C05443=1098.967,27.452,444.995,176.228,15.026,151.970
C05444=1098.962,27.202,445.009,176.226,15.025,151.971
C05445=1098.956,26.952,445.024,176.224,15.025,151.971
C05446=1098.951,26.703,445.039,176.221,15.024,151.971
C05447=1098.944,26.454,445.054,176.219,15.023,151.972
C05448=1098.939,26.204,445.069,176.217,15.022,151.972
C05449=1098.933,25.955,445.084,176.215,15.022,151.972
C05450=1098.927,25.705,445.098,176.212,15.021,151.973
C05451=1098.922,25.455,445.113,176.210,15.020,151.973
C05452=1098.916,25.206,445.128,176.208,15.020,151.973
C05453=1098.910,24.957,445.143,176.206,15.019,151.974
C05454=1098.904,24.708,445.157,176.203,15.018,151.974
C05455=1098.899,24.458,445.172,176.201,15.018,151.974
C05456=1098.893,24.208,445.187,176.199,15.017,151.975
C05457=1098.887,23.959,445.201,176.197,15.016,151.975
C05458=1098.881,23.709,445.217,176.194,15.015,151.975
C05459=1098.876,23.460,445.231,176.192,15.015,151.976
C05460=1098.869,23.210,445.246,176.190,15.014,151.976
C05461=1098.863,22.961,445.260,176.188,15.013,151.976
C05462=1098.858,22.712,445.276,176.186,15.012,151.976
C05463=1098.852,22.461,445.290,176.183,15.012,151.977
C05464=1098.847,22.213,445.304,176.182,15.011,151.977
C05465=1098.841,21.963,445.320,176.180,15.010,151.977
C05466=1098.835,21.713,445.334,176.177,15.009,151.978
C05467=1098.830,21.464,445.348,176.175,15.009,151.978
C05468=1098.823,21.214,445.363,176.173,15.008,151.979
C05469=1098.819,20.964,445.378,176.171,15.008,151.979
C05470=1098.813,20.716,445.392,176.168,15.006,151.979
C05471=1098.806,20.466,445.407,176.166,15.006,151.979
C05472=1098.801,20.216,445.421,176.164,15.005,151.980
C05473=1098.795,19.967,445.436,176.162,15.005,151.980
C05474=1098.789,19.717,445.451,176.159,15.004,151.980
C05475=1098.784,19.468,445.465,176.157,15.003,151.981
C05476=1098.778,19.218,445.480,176.155,15.002,151.981
C05477=1098.772,18.969,445.495,176.153,15.002,151.981
C05478=1098.766,18.719,445.509,176.151,15.001,151.982
C05479=1098.760,18.470,445.523,176.149,15.000,151.982
C05480=1098.755,18.220,445.538,176.147,14.999,151.982
C05481=1098.749,17.970,445.553,176.145,14.999,151.983
C05482=1098.743,17.721,445.567,176.143,14.998,151.983
C05483=1098.738,17.472,445.581,176.140,14.997,151.983
C05484=1098.731,17.222,445.596,176.138,14.996,151.984
C05485=1098.726,16.973,445.610,176.136,14.996,151.984
C05486=1098.720,16.724,445.625,176.134,14.995,151.984
C05487=1098.714,16.473,445.639,176.131,14.994,151.985
C05488=1098.709,16.224,445.654,176.129,14.993,151.985
C05489=1098.702,15.952,445.669,176.127,14.993,151.985
C05490=1098.696,15.680,445.685,176.125,14.992,151.985
C05491=1098.690,15.408,445.700,176.123,14.991,151.986
C05492=1098.684,15.136,445.716,176.120,14.991,151.986
C05493=1098.678,14.886,445.731,176.118,14.989,151.986
C05494=1098.672,14.637,445.745,176.116,14.988,151.987
C05495=1098.666,14.388,445.759,176.114,14.988,151.987
C05496=1098.660,14.137,445.773,176.112,14.987,151.987
C05497=1098.655,13.889,445.788,176.109,14.986,151.988
C05498=1098.649,13.639,445.802,176.107,14.985,151.988
C05499=1098.643,13.389,445.817,176.105,14.985,151.988
C05500=1098.637,13.140,445.831,176.103,14.984,151.989
C05501=1098.631,12.891,445.845,176.101,14.984,151.989
C05502=1098.625,12.640,445.860,176.098,14.983,151.989
C05503=1098.620,12.391,445.873,176.097,14.982,151.990
C05504=1098.614,12.142,445.888,176.095,14.981,151.990
C05505=1098.608,11.892,445.902,176.092,14.981,151.990
C05506=1098.602,11.642,445.915,176.091,14.980,151.990
C05507=1098.596,11.393,445.930,176.088,14.979,151.991
C05508=1098.590,11.143,445.944,176.086,14.978,151.991
C05509=1098.584,10.894,445.959,176.084,14.978,151.991
C05510=1098.579,10.645,445.973,176.082,14.977,151.992
C05511=1098.573,10.394,445.987,176.080,14.976,151.992
C05512=1098.567,10.145,446.002,176.077,14.975,151.992
C05513=1098.561,9.896,446.015,176.075,14.975,151.993
C05514=1098.556,9.646,446.029,176.073,14.974,151.993
C05515=1098.550,9.397,446.044,176.072,14.973,151.993
C05516=1098.543,9.147,446.057,176.070,14.972,151.993
C05517=1098.538,8.898,446.071,176.067,14.972,151.994
C05518=1098.532,8.648,446.085,176.065,14.971,151.994
C05519=1098.526,8.399,446.100,176.063,14.970,151.994
C05520=1098.520,8.149,446.114,176.061,14.969,151.995
C05521=1098.515,7.899,446.128,176.059,14.969,151.995
C05522=1098.510,7.650,446.142,176.056,14.968,151.995
C05523=1098.502,7.400,446.156,176.054,14.967,151.996
C05524=1098.497,7.151,446.170,176.052,14.966,151.996
C05525=1098.491,6.901,446.184,176.051,14.965,151.996
C05526=1098.486,6.652,446.198,176.048,14.965,151.997
C05527=1098.480,6.402,446.213,176.046,14.964,151.997
C05528=1098.474,6.153,446.227,176.044,14.963,151.997
C05529=1098.469,5.903,446.240,176.042,14.962,151.997
C05530=1098.462,5.654,446.254,176.040,14.962,151.998
C05531=1098.457,5.404,446.268,176.038,14.961,151.998
C05532=1098.451,5.154,446.282,176.036,14.961,151.998
C05533=1098.445,4.905,446.296,176.033,14.959,151.999
C05534=1098.440,4.655,446.310,176.031,14.958,151.999
C05535=1098.433,4.406,446.323,176.030,14.958,151.999
C05536=1098.428,4.156,446.337,176.028,14.957,151.999
C05537=1098.422,3.907,446.351,176.026,14.956,152.000
C05538=1098.416,3.657,446.365,176.023,14.955,152.000
C05539=1098.411,3.408,446.380,176.021,14.955,152.000
C05540=1098.404,3.158,446.393,176.019,14.954,152.001
C05541=1098.399,2.909,446.407,176.017,14.953,152.001
C05542=1098.393,2.659,446.421,176.015,14.952,152.001
C05543=1098.388,2.410,446.435,176.014,14.952,152.001
C05544=1098.382,2.160,446.449,176.011,14.950,152.002
C05545=1098.376,1.910,446.462,176.009,14.950,152.002
C05546=1098.370,1.661,446.476,176.007,14.949,152.002
C05547=1098.365,1.411,446.490,176.005,14.949,152.003
C05548=1098.359,1.161,446.504,176.003,14.948,152.003
C05549=1098.353,0.912,446.517,176.001,14.947,152.003
C05550=1098.348,0.663,446.531,175.998,14.946,152.003
C05551=1098.342,0.413,446.545,175.997,14.945,152.004
C05552=1098.337,0.163,446.559,175.995,14.944,152.004
C05553=1098.330,-0.107,446.574,175.993,14.943,152.004
C05554=1098.324,-0.377,446.588,175.990,14.942,152.004
C05555=1098.317,-0.646,446.604,175.988,14.941,152.005
C05556=1098.311,-0.917,446.619,175.986,14.941,152.005
C05557=1098.305,-1.166,446.632,175.983,14.940,152.005
C05558=1098.300,-1.416,446.646,175.982,14.939,152.006
C05559=1098.294,-1.665,446.660,175.980,14.938,152.006
C05560=1098.289,-1.915,446.673,175.978,14.938,152.006
C05561=1098.283,-2.165,446.686,175.976,14.937,152.006
C05562=1098.277,-2.414,446.700,175.974,14.936,152.007
C05563=1098.272,-2.664,446.714,175.971,14.935,152.007
C05564=1098.265,-2.913,446.727,175.970,14.934,152.007
C05565=1098.260,-3.163,446.741,175.968,14.933,152.007
C05566=1098.255,-3.412,446.755,175.966,14.932,152.008
C05567=1098.248,-3.661,446.768,175.964,14.932,152.008
C05568=1098.242,-3.912,446.782,175.962,14.931,152.008
C05569=1098.236,-4.161,446.796,175.960,14.930,152.008
C05570=1098.231,-4.411,446.810,175.957,14.929,152.009
C05571=1098.225,-4.660,446.822,175.955,14.929,152.009
C05572=1098.219,-4.910,446.836,175.953,14.928,152.009
C05573=1098.213,-5.159,446.849,175.952,14.927,152.010
C05574=1098.207,-5.409,446.863,175.950,14.926,152.010
C05575=1098.201,-5.658,446.876,175.948,14.926,152.010
C05576=1098.196,-5.908,446.890,175.946,14.925,152.010
C05577=1098.190,-6.157,446.904,175.943,14.924,152.011
C05578=1098.184,-6.408,446.917,175.941,14.923,152.011
C05579=1098.178,-6.657,446.930,175.940,14.922,152.011
C05580=1098.172,-6.907,446.944,175.938,14.921,152.012
C05581=1098.166,-7.156,446.958,175.935,14.921,152.012
C05582=1098.160,-7.406,446.971,175.934,14.920,152.012
C05583=1098.155,-7.655,446.984,175.932,14.920,152.013
C05584=1098.149,-7.905,446.998,175.930,14.919,152.013
C05585=1098.143,-8.154,447.011,175.927,14.917,152.013
C05586=1098.137,-8.404,447.025,175.925,14.917,152.013
C05587=1098.131,-8.653,447.038,175.923,14.916,152.014
C05588=1098.126,-8.903,447.051,175.922,14.915,152.014
C05589=1098.120,-9.153,447.065,175.920,14.915,152.014
C05590=1098.114,-9.402,447.078,175.918,14.914,152.014
C05591=1098.108,-9.652,447.091,175.916,14.913,152.015
C05592=1098.102,-9.901,447.104,175.914,14.912,152.015
C05593=1098.097,-10.151,447.118,175.911,14.911,152.015
C05594=1098.090,-10.400,447.131,175.909,14.910,152.015
C05595=1098.085,-10.650,447.145,175.908,14.909,152.016
C05596=1098.079,-10.900,447.158,175.906,14.909,152.016
C05597=1098.074,-11.149,447.172,175.904,14.908,152.016
C05598=1098.068,-11.399,447.184,175.902,14.907,152.016
C05599=1098.061,-11.648,447.198,175.900,14.906,152.017
C05600=1098.056,-11.898,447.211,175.898,14.906,152.017
C05601=1098.050,-12.148,447.224,175.896,14.904,152.017
C05602=1098.045,-12.397,447.238,175.894,14.904,152.018
C05603=1098.038,-12.647,447.251,175.892,14.903,152.018
C05604=1098.033,-12.896,447.264,175.890,14.902,152.018
C05605=1098.027,-13.146,447.278,175.888,14.901,152.018
C05606=1098.021,-13.396,447.290,175.886,14.901,152.019
C05607=1098.016,-13.645,447.304,175.884,14.900,152.019
C05608=1098.009,-13.895,447.317,175.882,14.899,152.019
C05609=1098.004,-14.144,447.329,175.881,14.898,152.019
C05610=1097.999,-14.393,447.343,175.878,14.897,152.020
C05611=1097.993,-14.643,447.356,175.876,14.896,152.020
C05612=1097.987,-14.893,447.369,175.874,14.896,152.020
C05613=1097.981,-15.143,447.382,175.872,14.895,152.020
C05614=1097.975,-15.392,447.395,175.870,14.894,152.021
C05615=1097.969,-15.641,447.409,175.868,14.893,152.021
C05616=1097.963,-15.891,447.421,175.867,14.893,152.021
C05617=1097.957,-16.160,447.436,175.865,14.892,152.021
C05618=1097.950,-16.428,447.449,175.862,14.891,152.022
C05619=1097.944,-16.697,447.464,175.860,14.890,152.022
C05620=1097.938,-16.965,447.477,175.858,14.890,152.022
C05621=1097.932,-17.214,447.491,175.856,14.889,152.023
C05622=1097.927,-17.465,447.504,175.854,14.888,152.023
C05623=1097.920,-17.714,447.517,175.852,14.887,152.023
C05624=1097.914,-17.964,447.530,175.850,14.886,152.023
C05625=1097.908,-18.213,447.543,175.848,14.885,152.024
C05626=1097.902,-18.463,447.556,175.846,14.885,152.024
C05627=1097.897,-18.712,447.569,175.844,14.884,152.024
C05628=1097.892,-18.962,447.582,175.842,14.883,152.025
C05629=1097.885,-19.211,447.595,175.840,14.882,152.025
C05630=1097.879,-19.461,447.607,175.838,14.882,152.025
C05631=1097.873,-19.710,447.621,175.837,14.881,152.025
C05632=1097.867,-19.960,447.633,175.835,14.880,152.026
C05633=1097.862,-20.210,447.646,175.833,14.879,152.026
C05634=1097.856,-20.459,447.660,175.831,14.879,152.026
C05635=1097.850,-20.709,447.672,175.829,14.878,152.026
C05636=1097.844,-20.959,447.685,175.827,14.877,152.026
C05637=1097.839,-21.208,447.698,175.825,14.875,152.027
C05638=1097.833,-21.458,447.710,175.823,14.875,152.027
C05639=1097.827,-21.707,447.724,175.821,14.874,152.027
C05640=1097.821,-21.957,447.737,175.819,14.873,152.027
C05641=1097.815,-22.206,447.750,175.817,14.872,152.028
C05642=1097.809,-22.456,447.762,175.815,14.872,152.028
C05643=1097.803,-22.706,447.775,175.814,14.871,152.028
C05644=1097.798,-22.955,447.788,175.812,14.870,152.029
C05645=1097.792,-23.205,447.800,175.810,14.869,152.029
C05646=1097.786,-23.455,447.813,175.808,14.869,152.029
C05647=1097.780,-23.704,447.827,175.806,14.868,152.029
C05648=1097.774,-23.954,447.839,175.804,14.867,152.030
C05649=1097.768,-24.204,447.852,175.802,14.866,152.030
C05650=1097.763,-24.453,447.864,175.800,14.866,152.030
C05651=1097.757,-24.702,447.877,175.798,14.864,152.030
C05652=1097.751,-24.952,447.890,175.796,14.864,152.031
C05653=1097.745,-25.202,447.903,175.794,14.863,152.031
C05654=1097.739,-25.451,447.916,175.792,14.862,152.031
C05655=1097.734,-25.701,447.928,175.790,14.861,152.031
C05656=1097.728,-25.951,447.941,175.789,14.860,152.032
C05657=1097.723,-26.201,447.954,175.787,14.859,152.032
C05658=1097.717,-26.450,447.966,175.785,14.859,152.032
C05659=1097.710,-26.700,447.980,175.783,14.858,152.032
C05660=1097.705,-26.949,447.992,175.781,14.857,152.033
C05661=1097.699,-27.199,448.004,175.779,14.857,152.033
C05662=1097.693,-27.449,448.017,175.777,14.856,152.033
C05663=1097.687,-27.698,448.030,175.776,14.855,152.033
C05664=1097.681,-27.948,448.043,175.774,14.854,152.034
C05665=1097.676,-28.197,448.055,175.772,14.854,152.034
C05666=1097.669,-28.447,448.067,175.770,14.853,152.034
C05667=1097.663,-28.696,448.079,175.768,14.852,152.034
C05668=1097.657,-28.946,448.093,175.766,14.851,152.035
C05669=1097.651,-29.196,448.105,175.764,14.851,152.035
C05670=1097.646,-29.445,448.117,175.762,14.850,152.035
C05671=1097.640,-29.695,448.130,175.760,14.849,152.035
C05672=1097.634,-29.945,448.142,175.759,14.848,152.036
C05673=1097.628,-30.194,448.155,175.757,14.848,152.036
C05674=1097.622,-30.444,448.168,175.754,14.846,152.036
C05675=1097.617,-30.693,448.181,175.752,14.846,152.036
C05676=1097.611,-30.943,448.193,175.750,14.845,152.037
C05677=1097.604,-31.192,448.205,175.748,14.844,152.037
C05678=1097.598,-31.442,448.218,175.747,14.843,152.037
C05679=1097.593,-31.691,448.230,175.745,14.842,152.037
C05680=1097.587,-31.941,448.242,175.743,14.841,152.038
C05681=1097.581,-32.209,448.256,175.741,14.841,152.038
C05682=1097.575,-32.477,448.269,175.739,14.840,152.038
C05683=1097.567,-32.744,448.283,175.737,14.839,152.038
C05684=1097.561,-33.012,448.296,175.736,14.839,152.039
C05685=1097.556,-33.261,448.308,175.734,14.838,152.039
C05686=1097.550,-33.511,448.320,175.732,14.837,152.039
C05687=1097.544,-33.761,448.333,175.730,14.836,152.039
C05688=1097.538,-34.010,448.346,175.728,14.836,152.040
C05689=1097.532,-34.259,448.358,175.726,14.835,152.040
C05690=1097.526,-34.509,448.370,175.724,14.834,152.040
C05691=1097.520,-34.759,448.383,175.722,14.833,152.040
C05692=1097.515,-35.008,448.395,175.721,14.833,152.041
C05693=1097.509,-35.258,448.408,175.719,14.832,152.041
C05694=1097.503,-35.508,448.420,175.717,14.831,152.041
C05695=1097.497,-35.758,448.431,175.715,14.830,152.042
C05696=1097.492,-36.007,448.444,175.713,14.830,152.042
C05697=1097.486,-36.257,448.456,175.711,14.829,152.042
C05698=1097.480,-36.507,448.469,175.709,14.827,152.042
C05699=1097.474,-36.756,448.481,175.707,14.826,152.042
C05700=1097.468,-37.006,448.493,175.705,14.826,152.043
C05701=1097.462,-37.256,448.505,175.703,14.825,152.043
C05702=1097.457,-37.505,448.518,175.701,14.824,152.043
C05703=1097.451,-37.755,448.530,175.699,14.823,152.044
C05704=1097.445,-38.005,448.543,175.698,14.823,152.044
C05705=1097.439,-38.254,448.555,175.696,14.822,152.044
C05706=1097.433,-38.503,448.567,175.695,14.822,152.044
C05707=1097.427,-38.753,448.579,175.693,14.821,152.044
C05708=1097.422,-39.003,448.592,175.691,14.820,152.045
C05709=1097.415,-39.253,448.603,175.689,14.819,152.045
C05710=1097.409,-39.503,448.615,175.687,14.818,152.045
C05711=1097.404,-39.752,448.628,175.685,14.818,152.045
C05712=1097.397,-40.001,448.640,175.684,14.817,152.046
C05713=1097.391,-40.251,448.652,175.682,14.816,152.046
C05714=1097.386,-40.500,448.664,175.680,14.816,152.046
C05715=1097.379,-40.750,448.676,175.678,14.815,152.046
C05716=1097.374,-41.000,448.688,175.676,14.814,152.047
C05717=1097.369,-41.250,448.700,175.674,14.813,152.047
C05718=1097.362,-41.499,448.712,175.672,14.813,152.047
C05719=1097.356,-41.749,448.725,175.670,14.812,152.047
C05720=1097.350,-41.998,448.736,175.669,14.811,152.048
C05721=1097.344,-42.248,448.749,175.667,14.810,152.048
C05722=1097.338,-42.498,448.761,175.665,14.810,152.048
C05723=1097.332,-42.747,448.772,175.663,14.809,152.049
C05724=1097.326,-42.997,448.785,175.661,14.808,152.049
C05725=1097.321,-43.247,448.797,175.659,14.807,152.049
C05726=1097.315,-43.497,448.808,175.657,14.807,152.049
C05727=1097.309,-43.746,448.821,175.656,14.806,152.049
C05728=1097.303,-43.995,448.832,175.654,14.805,152.050
C05729=1097.297,-44.245,448.845,175.652,14.804,152.050
C05730=1097.291,-44.496,448.857,175.650,14.803,152.050
C05731=1097.285,-44.745,448.868,175.648,14.803,152.050
C05732=1097.279,-44.994,448.881,175.646,14.802,152.051
C05733=1097.273,-45.243,448.893,175.644,14.801,152.051
C05734=1097.268,-45.494,448.904,175.643,14.800,152.051
C05735=1097.261,-45.743,448.916,175.641,14.800,152.052
C05736=1097.256,-45.993,448.929,175.639,14.799,152.052
C05737=1097.250,-46.243,448.940,175.637,14.798,152.052
C05738=1097.244,-46.492,448.952,175.635,14.797,152.052
C05739=1097.238,-46.742,448.965,175.634,14.797,152.053
C05740=1097.232,-46.992,448.976,175.632,14.797,152.053
C05741=1097.227,-47.241,448.988,175.630,14.795,152.053
C05742=1097.220,-47.491,449.000,175.629,14.795,152.053
C05743=1097.215,-47.741,449.011,175.627,14.794,152.053
C05744=1097.208,-47.990,449.023,175.625,14.793,152.054
C05745=1097.202,-48.258,449.036,175.623,14.792,152.054
C05746=1097.196,-48.526,449.049,175.621,14.792,152.054
C05747=1097.190,-48.794,449.062,175.619,14.791,152.054
C05748=1097.183,-49.061,449.074,175.616,14.790,152.055
C05749=1097.178,-49.312,449.086,175.615,14.790,152.055
C05750=1097.172,-49.561,449.098,175.614,14.789,152.055
C05751=1097.166,-49.810,449.110,175.612,14.788,152.055
C05752=1097.160,-50.060,449.121,175.610,14.787,152.056
C05753=1097.154,-50.310,449.134,175.608,14.787,152.056
C05754=1097.148,-50.559,449.145,175.606,14.786,152.056
C05755=1097.142,-50.809,449.157,175.604,14.785,152.057
C05756=1097.136,-51.059,449.168,175.602,14.784,152.057
C05757=1097.130,-51.308,449.180,175.600,14.784,152.057
C05758=1097.124,-51.558,449.193,175.598,14.783,152.057
C05759=1097.118,-51.808,449.203,175.597,14.782,152.058
C05760=1097.112,-52.057,449.215,175.595,14.782,152.058
C05761=1097.106,-52.308,449.227,175.593,14.781,152.058
C05762=1097.100,-52.557,449.239,175.592,14.781,152.058
C05763=1097.094,-52.807,449.250,175.590,14.780,152.059
C05764=1097.089,-53.056,449.262,175.588,14.779,152.059
C05765=1097.082,-53.306,449.273,175.586,14.778,152.059
C05766=1097.076,-53.555,449.285,175.584,14.778,152.059
C05767=1097.070,-53.805,449.296,175.582,14.777,152.060
C05768=1097.064,-54.055,449.309,175.580,14.776,152.060
C05769=1097.058,-54.305,449.320,175.579,14.776,152.060
C05770=1097.051,-54.554,449.332,175.577,14.775,152.060
C05771=1097.046,-54.804,449.343,175.575,14.774,152.061
C05772=1097.040,-55.054,449.355,175.573,14.773,152.061
C05773=1097.034,-55.303,449.366,175.572,14.773,152.061
C05774=1097.027,-55.553,449.378,175.570,14.773,152.061
C05775=1097.022,-55.802,449.389,175.568,14.772,152.062
C05776=1097.016,-56.052,449.401,175.566,14.771,152.062
C05777=1097.010,-56.301,449.412,175.564,14.770,152.062
C05778=1097.004,-56.552,449.424,175.562,14.770,152.063
C05779=1096.998,-56.801,449.435,175.561,14.769,152.063
C05780=1096.992,-57.051,449.447,175.559,14.768,152.063
C05781=1096.986,-57.300,449.459,175.557,14.767,152.063
C05782=1096.980,-57.550,449.470,175.556,14.767,152.064
C05783=1096.974,-57.799,449.481,175.554,14.767,152.064
C05784=1096.968,-58.049,449.493,175.552,14.766,152.064
C05785=1096.962,-58.299,449.504,175.550,14.765,152.064
C05786=1096.956,-58.549,449.516,175.548,14.764,152.064
C05787=1096.950,-58.798,449.527,175.547,14.763,152.065
C05788=1096.944,-59.048,449.538,175.545,14.762,152.065
C05789=1096.938,-59.297,449.550,175.543,14.762,152.065
C05790=1096.932,-59.548,449.562,175.542,14.762,152.065
C05791=1096.926,-59.797,449.573,175.540,14.761,152.066
C05792=1096.920,-60.047,449.584,175.538,14.760,152.066
C05793=1096.914,-60.296,449.595,175.536,14.759,152.066
C05794=1096.908,-60.547,449.607,175.534,14.759,152.066
C05795=1096.902,-60.796,449.619,175.532,14.758,152.067
C05796=1096.896,-61.046,449.630,175.530,14.757,152.067
C05797=1096.890,-61.295,449.641,175.529,14.757,152.067
C05798=1096.884,-61.544,449.652,175.527,14.756,152.068
C05799=1096.878,-61.794,449.664,175.526,14.756,152.068
C05800=1096.873,-62.044,449.675,175.524,14.755,152.068
C05801=1096.866,-62.294,449.686,175.522,14.754,152.068
C05802=1096.860,-62.543,449.698,175.520,14.753,152.069
C05803=1096.855,-62.793,449.709,175.518,14.753,152.069
C05804=1096.848,-63.043,449.720,175.516,14.752,152.069
C05805=1096.842,-63.292,449.731,175.515,14.752,152.069
C05806=1096.837,-63.542,449.744,175.513,14.751,152.070
C05807=1096.831,-63.792,449.754,175.511,14.750,152.070
C05808=1096.825,-64.042,449.766,175.509,14.750,152.070
C05809=1096.818,-64.310,449.777,175.507,14.749,152.070
C05810=1096.812,-64.579,449.790,175.506,14.748,152.071
C05811=1096.805,-64.849,449.801,175.504,14.748,152.071
C05812=1096.799,-65.118,449.814,175.502,14.747,152.071
C05813=1096.793,-65.368,449.825,175.500,14.746,152.071
C05814=1096.787,-65.618,449.836,175.498,14.745,152.072
C05815=1096.781,-65.867,449.848,175.496,14.745,152.072
C05816=1096.775,-66.117,449.859,175.495,14.745,152.072
C05817=1096.770,-66.367,449.871,175.493,14.744,152.072
C05818=1096.764,-66.616,449.881,175.491,14.743,152.073
C05819=1096.758,-66.866,449.893,175.489,14.742,152.073
C05820=1096.752,-67.116,449.904,175.488,14.742,152.073
C05821=1096.746,-67.365,449.914,175.486,14.741,152.074
C05822=1096.740,-67.615,449.926,175.485,14.741,152.074
C05823=1096.734,-67.865,449.937,175.483,14.740,152.074
C05824=1096.728,-68.114,449.948,175.481,14.739,152.074
C05825=1096.722,-68.364,449.959,175.479,14.739,152.075
C05826=1096.716,-68.614,449.970,175.477,14.738,152.075
C05827=1096.710,-68.863,449.981,175.475,14.737,152.075
C05828=1096.705,-69.114,449.993,175.474,14.737,152.075
C05829=1096.699,-69.363,450.004,175.472,14.736,152.076
C05830=1096.693,-69.613,450.015,175.470,14.736,152.076
C05831=1096.687,-69.863,450.026,175.468,14.735,152.076
C05832=1096.681,-70.112,450.038,175.467,14.734,152.076
C05833=1096.675,-70.361,450.048,175.465,14.733,152.077
C05834=1096.669,-70.611,450.059,175.464,14.733,152.077
C05835=1096.663,-70.861,450.071,175.462,14.733,152.077
C05836=1096.657,-71.110,450.081,175.460,14.732,152.077
C05837=1096.652,-71.360,450.092,175.458,14.731,152.078
C05838=1096.645,-71.610,450.104,175.456,14.730,152.078
C05839=1096.639,-71.860,450.114,175.455,14.730,152.078
C05840=1096.634,-72.109,450.125,175.453,14.730,152.078
C05841=1096.628,-72.359,450.136,175.451,14.729,152.079
C05842=1096.622,-72.609,450.147,175.450,14.728,152.079
C05843=1096.616,-72.858,450.158,175.448,14.727,152.079
C05844=1096.610,-73.108,450.169,175.446,14.726,152.079
C05845=1096.604,-73.357,450.180,175.445,14.726,152.079
C05846=1096.599,-73.608,450.192,175.443,14.725,152.080
C05847=1096.593,-73.857,450.203,175.441,14.725,152.080
C05848=1096.587,-74.107,450.214,175.439,14.724,152.080
C05849=1096.581,-74.356,450.224,175.437,14.723,152.081
C05850=1096.575,-74.606,450.235,175.436,14.723,152.081
C05851=1096.569,-74.856,450.246,175.434,14.722,152.081
C05852=1096.563,-75.106,450.256,175.432,14.722,152.081
C05853=1096.557,-75.356,450.267,175.430,14.721,152.082
C05854=1096.551,-75.605,450.278,175.429,14.721,152.082
C05855=1096.546,-75.855,450.289,175.427,14.720,152.082
C05856=1096.539,-76.105,450.300,175.425,14.720,152.082
C05857=1096.533,-76.354,450.311,175.423,14.719,152.083
C05858=1096.527,-76.604,450.322,175.421,14.718,152.083
C05859=1096.521,-76.853,450.333,175.420,14.718,152.083
C05860=1096.515,-77.103,450.344,175.418,14.717,152.084
C05861=1096.509,-77.353,450.355,175.417,14.717,152.084
C05862=1096.503,-77.602,450.366,175.415,14.716,152.084
C05863=1096.497,-77.851,450.376,175.414,14.716,152.084
C05864=1096.491,-78.102,450.386,175.412,14.715,152.085
C05865=1096.485,-78.352,450.397,175.410,14.714,152.085
C05866=1096.479,-78.601,450.408,175.408,14.714,152.085
C05867=1096.474,-78.851,450.419,175.406,14.713,152.085
C05868=1096.467,-79.101,450.430,175.405,14.713,152.086
C05869=1096.461,-79.350,450.440,175.403,14.712,152.086
C05870=1096.455,-79.600,450.451,175.401,14.712,152.086
C05871=1096.450,-79.850,450.462,175.399,14.711,152.087
C05872=1096.443,-80.100,450.473,175.398,14.711,152.087
C05873=1096.436,-80.371,450.484,175.396,14.710,152.087
C05874=1096.430,-80.642,450.495,175.394,14.710,152.087
C05875=1096.424,-80.914,450.507,175.392,14.709,152.088
C05876=1096.417,-81.185,450.518,175.390,14.709,152.088
C05877=1096.411,-81.434,450.529,175.388,14.708,152.088
C05878=1096.405,-81.685,450.541,175.387,14.708,152.088
C05879=1096.398,-81.934,450.551,175.385,14.707,152.089
C05880=1096.393,-82.184,450.561,175.383,14.706,152.089
C05881=1096.387,-82.433,450.572,175.381,14.706,152.089
C05882=1096.380,-82.683,450.582,175.380,14.706,152.089
C05883=1096.374,-82.933,450.593,175.378,14.705,152.090
C05884=1096.369,-83.183,450.604,175.376,14.705,152.090
C05885=1096.362,-83.432,450.614,175.374,14.704,152.090
C05886=1096.356,-83.682,450.625,175.373,14.704,152.091
C05887=1096.350,-83.932,450.636,175.371,14.703,152.091
C05888=1096.344,-84.182,450.645,175.369,14.702,152.091
C05889=1096.338,-84.431,450.656,175.368,14.702,152.091
C05890=1096.331,-84.681,450.667,175.366,14.702,152.092
C05891=1096.325,-84.930,450.678,175.364,14.701,152.092
C05892=1096.320,-85.181,450.688,175.362,14.701,152.092
C05893=1096.313,-85.430,450.698,175.361,14.700,152.093
C05894=1096.308,-85.679,450.709,175.359,14.700,152.093
C05895=1096.301,-85.930,450.719,175.357,14.699,152.093
C05896=1096.295,-86.179,450.730,175.356,14.698,152.093
C05897=1096.289,-86.429,450.741,175.354,14.699,152.094
C05898=1096.283,-86.679,450.750,175.352,14.698,152.094
C05899=1096.278,-86.928,450.761,175.350,14.697,152.094
C05900=1096.270,-87.178,450.772,175.348,14.696,152.095
C05901=1096.265,-87.428,450.782,175.347,14.696,152.095
C05902=1096.259,-87.677,450.793,175.346,14.696,152.095
C05903=1096.253,-87.927,450.803,175.344,14.695,152.095
C05904=1096.247,-88.177,450.813,175.342,14.695,152.096
C05905=1096.240,-88.427,450.824,175.340,14.695,152.096
C05906=1096.235,-88.676,450.835,175.338,14.694,152.096
C05907=1096.228,-88.926,450.845,175.337,14.694,152.097
C05908=1096.223,-89.175,450.855,175.335,14.693,152.097
C05909=1096.217,-89.426,450.866,175.334,14.692,152.097
C05910=1096.211,-89.675,450.876,175.332,14.692,152.097
C05911=1096.205,-89.924,450.887,175.330,14.692,152.098
C05912=1096.198,-90.175,450.897,175.328,14.691,152.098
C05913=1096.193,-90.424,450.908,175.326,14.691,152.098
C05914=1096.186,-90.674,450.917,175.325,14.690,152.098
C05915=1096.181,-90.923,450.928,175.323,14.690,152.099
C05916=1096.174,-91.173,450.938,175.322,14.689,152.099
C05917=1096.169,-91.423,450.948,175.320,14.689,152.099
C05918=1096.162,-91.672,450.959,175.318,14.689,152.100
C05919=1096.157,-91.922,450.969,175.316,14.688,152.100
C05920=1096.150,-92.172,450.980,175.315,14.687,152.100
C05921=1096.144,-92.422,450.990,175.313,14.687,152.100
C05922=1096.139,-92.672,451.001,175.312,14.686,152.101
C05923=1096.132,-92.921,451.010,175.309,14.686,152.101
C05924=1096.127,-93.171,451.021,175.308,14.686,152.101
C05925=1096.120,-93.421,451.031,175.306,14.685,152.102
C05926=1096.115,-93.670,451.041,175.304,14.685,152.102
C05927=1096.109,-93.920,451.051,175.303,14.684,152.102
C05928=1096.103,-94.169,451.062,175.301,14.684,152.102
C05929=1096.097,-94.419,451.072,175.299,14.684,152.103
C05930=1096.091,-94.669,451.082,175.298,14.683,152.103
C05931=1096.084,-94.919,451.092,175.296,14.683,152.103
C05932=1096.079,-95.169,451.102,175.294,14.682,152.104
C05933=1096.072,-95.418,451.113,175.293,14.682,152.104
C05934=1096.067,-95.669,451.123,175.291,14.681,152.104
C05935=1096.060,-95.918,451.133,175.289,14.681,152.104
C05936=1096.055,-96.168,451.143,175.288,14.681,152.105
C05937=1096.048,-96.441,451.155,175.286,14.680,152.105
C05938=1096.042,-96.714,451.166,175.284,14.679,152.105
C05939=1096.035,-96.988,451.176,175.282,14.679,152.106
C05940=1096.028,-97.262,451.187,175.280,14.678,152.106
C05941=1096.022,-97.512,451.198,175.279,14.678,152.106
C05942=1096.016,-97.762,451.208,175.277,14.678,152.106
C05943=1096.011,-98.012,451.218,175.275,14.677,152.107
C05944=1096.004,-98.261,451.228,175.274,14.677,152.107
C05945=1095.998,-98.511,451.238,175.272,14.677,152.107
C05946=1095.992,-98.761,451.249,175.270,14.676,152.108
C05947=1095.986,-99.011,451.259,175.269,14.676,152.108
C05948=1095.980,-99.260,451.268,175.267,14.675,152.108
C05949=1095.974,-99.510,451.279,175.266,14.675,152.109
C05950=1095.968,-99.760,451.289,175.263,14.675,152.109
C05951=1095.961,-100.009,451.298,175.262,14.674,152.109
C05952=1095.955,-100.259,451.308,175.260,14.674,152.109
C05953=1095.950,-100.509,451.319,175.259,14.674,152.110
C05954=1095.943,-100.759,451.328,175.256,14.673,152.110
C05955=1095.937,-101.008,451.339,175.255,14.673,152.110
C05956=1095.931,-101.258,451.349,175.253,14.673,152.111
C05957=1095.925,-101.508,451.358,175.252,14.672,152.111
C05958=1095.919,-101.757,451.369,175.250,14.672,152.111
C05959=1095.913,-102.007,451.379,175.248,14.671,152.112
C05960=1095.907,-102.257,451.388,175.247,14.671,152.112
C05961=1095.901,-102.506,451.399,175.245,14.671,152.112
C05962=1095.895,-102.756,451.408,175.243,14.670,152.112
C05963=1095.889,-103.006,451.418,175.242,14.670,152.113
C05964=1095.883,-103.255,451.429,175.240,14.670,152.113
C05965=1095.876,-103.505,451.438,175.239,14.670,152.113
C05966=1095.870,-103.755,451.448,175.237,14.669,152.114
C05967=1095.864,-104.005,451.458,175.235,14.669,152.114
C05968=1095.858,-104.255,451.468,175.233,14.669,152.114
C05969=1095.852,-104.504,451.478,175.232,14.668,152.115
C05970=1095.845,-104.754,451.488,175.230,14.668,152.115
C05971=1095.840,-105.004,451.498,175.229,14.667,152.115
C05972=1095.834,-105.253,451.508,175.226,14.667,152.115
C05973=1095.827,-105.503,451.518,175.225,14.667,152.116
C05974=1095.821,-105.753,451.527,175.223,14.666,152.116
C05975=1095.816,-106.003,451.537,175.221,14.666,152.116
C05976=1095.810,-106.253,451.547,175.220,14.666,152.117
C05977=1095.803,-106.502,451.557,175.218,14.665,152.117
C05978=1095.797,-106.752,451.567,175.217,14.666,152.117
C05979=1095.791,-107.002,451.576,175.215,14.665,152.118
C05980=1095.785,-107.251,451.586,175.213,14.664,152.118
C05981=1095.780,-107.501,451.596,175.211,14.665,152.118
C05982=1095.773,-107.750,451.606,175.210,14.664,152.118
C05983=1095.767,-108.000,451.616,175.208,14.664,152.119
C05984=1095.761,-108.250,451.625,175.206,14.664,152.119
C05985=1095.755,-108.500,451.635,175.205,14.663,152.119
C05986=1095.749,-108.749,451.644,175.203,14.663,152.120
C05987=1095.742,-108.999,451.654,175.201,14.663,152.120
C05988=1095.737,-109.249,451.665,175.200,14.662,152.120
C05989=1095.731,-109.498,451.674,175.198,14.662,152.121
C05990=1095.724,-109.748,451.684,175.197,14.662,152.121
C05991=1095.718,-109.998,451.693,175.195,14.661,152.121
C05992=1095.712,-110.248,451.703,175.193,14.661,152.122
C05993=1095.706,-110.498,451.713,175.191,14.661,152.122
C05994=1095.700,-110.747,451.722,175.190,14.660,152.122
C05995=1095.693,-110.997,451.732,175.188,14.661,152.123
C05996=1095.687,-111.247,451.741,175.186,14.660,152.123
C05997=1095.681,-111.496,451.752,175.185,14.660,152.123
C05998=1095.675,-111.746,451.761,175.183,14.660,152.123
C05999=1095.668,-111.996,451.771,175.181,14.659,152.124
C06000=1095.663,-112.246,451.781,175.180,14.659,152.124
C06001=1095.656,-112.509,451.791,175.178,14.659,152.124
C06002=1095.650,-112.774,451.801,175.176,14.659,152.125
C06003=1095.643,-113.037,451.811,175.174,14.658,152.125
C06004=1095.637,-113.301,451.821,175.173,14.658,152.125
C06005=1095.631,-113.550,451.831,175.171,14.658,152.126
C06006=1095.625,-113.800,451.840,175.169,14.657,152.126
C06007=1095.619,-114.050,451.850,175.168,14.658,152.126
C06008=1095.613,-114.300,451.859,175.166,14.657,152.127
C06009=1095.606,-114.550,451.869,175.165,14.657,152.127
C06010=1095.600,-114.799,451.879,175.163,14.657,152.127
C06011=1095.595,-115.049,451.888,175.161,14.656,152.128
C06012=1095.588,-115.298,451.897,175.159,14.656,152.128
C06013=1095.582,-115.548,451.907,175.157,14.656,152.128
C06014=1095.576,-115.798,451.917,175.156,14.656,152.129
C06015=1095.570,-116.048,451.926,175.154,14.655,152.129
C06016=1095.564,-116.298,451.936,175.153,14.655,152.129
C06017=1095.558,-116.547,451.945,175.151,14.655,152.130
C06018=1095.551,-116.797,451.955,175.150,14.655,152.130
C06019=1095.545,-117.047,451.964,175.147,14.655,152.130
C06020=1095.539,-117.297,451.974,175.146,14.654,152.130
C06021=1095.533,-117.546,451.983,175.144,14.654,152.131
C06022=1095.526,-117.796,451.992,175.143,14.654,152.131
C06023=1095.520,-118.045,452.002,175.141,14.654,152.132
C06024=1095.514,-118.295,452.011,175.139,14.653,152.132
C06025=1095.508,-118.545,452.021,175.137,14.654,152.132
C06026=1095.502,-118.794,452.030,175.136,14.653,152.132
C06027=1095.496,-119.044,452.040,175.134,14.653,152.133
C06028=1095.490,-119.294,452.049,175.132,14.653,152.133
C06029=1095.483,-119.544,452.059,175.131,14.652,152.133
C06030=1095.477,-119.794,452.069,175.129,14.652,152.134
C06031=1095.471,-120.044,452.077,175.128,14.652,152.134
C06032=1095.465,-120.294,452.087,175.126,14.652,152.134
C06033=1095.459,-120.543,452.096,175.125,14.652,152.135
C06034=1095.453,-120.792,452.105,175.122,14.652,152.135
C06035=1095.447,-121.042,452.115,175.121,14.651,152.135
C06036=1095.440,-121.292,452.124,175.119,14.651,152.136
C06037=1095.434,-121.542,452.134,175.118,14.651,152.136
C06038=1095.428,-121.792,452.143,175.116,14.651,152.136
C06039=1095.422,-122.042,452.152,175.115,14.651,152.137
C06040=1095.416,-122.292,452.162,175.112,14.651,152.137
C06041=1095.410,-122.541,452.171,175.111,14.651,152.137
C06042=1095.404,-122.790,452.180,175.109,14.650,152.138
C06043=1095.397,-123.040,452.190,175.108,14.650,152.138
C06044=1095.391,-123.290,452.199,175.106,14.650,152.138
C06045=1095.385,-123.540,452.208,175.105,14.650,152.139
C06046=1095.379,-123.790,452.218,175.102,14.650,152.139
C06047=1095.374,-124.039,452.227,175.101,14.650,152.139
C06048=1095.367,-124.289,452.236,175.099,14.649,152.140
C06049=1095.361,-124.539,452.245,175.098,14.649,152.140
C06050=1095.354,-124.788,452.255,175.096,14.649,152.140
C06051=1095.348,-125.039,452.264,175.095,14.649,152.141
C06052=1095.342,-125.289,452.273,175.092,14.649,152.141
C06053=1095.335,-125.538,452.282,175.091,14.649,152.141
C06054=1095.330,-125.787,452.292,175.089,14.648,152.142
C06055=1095.324,-126.038,452.300,175.088,14.649,152.142
C06056=1095.318,-126.287,452.310,175.086,14.648,152.142
C06057=1095.311,-126.537,452.319,175.084,14.648,152.143
C06058=1095.305,-126.787,452.328,175.083,14.648,152.143
C06059=1095.299,-127.037,452.338,175.081,14.648,152.143
C06060=1095.293,-127.286,452.346,175.079,14.648,152.144
C06061=1095.286,-127.548,452.356,175.078,14.648,152.144
C06062=1095.279,-127.809,452.365,175.076,14.648,152.145
C06063=1095.273,-128.070,452.376,175.074,14.648,152.145
C06064=1095.273,-128.332,452.387,175.073,14.646,152.145
C06065=1094.865,-128.352,452.276,175.028,14.753,152.175
C06066=1094.864,-128.093,452.264,175.029,14.755,152.175
C06067=1094.871,-127.831,452.255,175.031,14.756,152.175
C06068=1094.877,-127.570,452.246,175.033,14.755,152.175
C06069=1094.883,-127.309,452.236,175.034,14.756,152.174
C06070=1094.890,-127.059,452.227,175.036,14.756,152.174
C06071=1094.896,-126.809,452.217,175.038,14.756,152.174
C06072=1094.902,-126.559,452.208,175.039,14.756,152.173
C06073=1094.908,-126.310,452.199,175.041,14.756,152.173
C06074=1094.915,-126.060,452.190,175.043,14.756,152.173
C06075=1094.921,-125.810,452.181,175.045,14.757,152.172
C06076=1094.927,-125.561,452.171,175.046,14.757,152.172
C06077=1094.933,-125.311,452.162,175.048,14.757,152.172
C06078=1094.940,-125.061,452.153,175.049,14.757,152.171
C06079=1094.946,-124.811,452.144,175.051,14.757,152.171
C06080=1094.951,-124.562,452.135,175.052,14.757,152.171
C06081=1094.958,-124.312,452.125,175.055,14.758,152.170
C06082=1094.964,-124.062,452.115,175.056,14.758,152.170
C06083=1094.970,-123.812,452.107,175.058,14.758,152.170
C06084=1094.977,-123.562,452.098,175.059,14.758,152.169
C06085=1094.983,-123.313,452.088,175.061,14.758,152.169
C06086=1094.988,-123.063,452.079,175.062,14.758,152.169
C06087=1094.994,-122.814,452.069,175.064,14.759,152.169
C06088=1095.001,-122.564,452.060,175.066,14.759,152.168
C06089=1095.007,-122.314,452.051,175.068,14.759,152.168
C06090=1095.013,-122.064,452.042,175.069,14.759,152.167
C06091=1095.020,-121.814,452.032,175.071,14.760,152.167
C06092=1095.026,-121.564,452.023,175.072,14.759,152.167
C06093=1095.032,-121.315,452.013,175.074,14.760,152.167
C06094=1095.037,-121.065,452.004,175.076,14.759,152.166
C06095=1095.044,-120.816,451.994,175.078,14.760,152.166
C06096=1095.050,-120.565,451.986,175.079,14.760,152.166
C06097=1095.056,-120.316,451.977,175.081,14.760,152.165
C06098=1095.063,-120.066,451.967,175.082,14.761,152.165
C06099=1095.069,-119.816,451.957,175.084,14.761,152.165
C06100=1095.075,-119.566,451.948,175.085,14.761,152.164
C06101=1095.081,-119.317,451.938,175.088,14.761,152.164
C06102=1095.087,-119.067,451.929,175.089,14.762,152.164
C06103=1095.093,-118.818,451.920,175.091,14.761,152.163
C06104=1095.099,-118.568,451.910,175.093,14.762,152.163
C06105=1095.105,-118.318,451.900,175.094,14.762,152.163
C06106=1095.111,-118.068,451.891,175.096,14.762,152.162
C06107=1095.118,-117.819,451.881,175.097,14.763,152.162
C06108=1095.123,-117.568,451.872,175.099,14.763,152.162
C06109=1095.130,-117.319,451.863,175.100,14.763,152.161
C06110=1095.136,-117.069,451.854,175.102,14.764,152.161
C06111=1095.143,-116.819,451.844,175.104,14.763,152.161
C06112=1095.148,-116.570,451.835,175.106,14.764,152.161
C06113=1095.154,-116.320,451.826,175.107,14.764,152.160
C06114=1095.161,-116.070,451.816,175.109,14.764,152.160
C06115=1095.167,-115.821,451.806,175.111,14.765,152.160
C06116=1095.173,-115.571,451.797,175.112,14.765,152.159
C06117=1095.179,-115.321,451.787,175.114,14.765,152.159
C06118=1095.185,-115.071,451.778,175.116,14.765,152.159
C06119=1095.191,-114.821,451.768,175.118,14.766,152.158
C06120=1095.198,-114.572,451.759,175.119,14.766,152.158
C06121=1095.204,-114.322,451.749,175.121,14.766,152.158
C06122=1095.210,-114.072,451.739,175.122,14.766,152.157
C06123=1095.216,-113.822,451.730,175.124,14.767,152.157
C06124=1095.222,-113.572,451.720,175.126,14.767,152.157
C06125=1095.228,-113.323,451.711,175.127,14.767,152.156
C06126=1095.234,-113.059,451.700,175.129,14.767,152.156
C06127=1095.241,-112.794,451.690,175.130,14.767,152.156
C06128=1095.248,-112.531,451.680,175.132,14.768,152.156
C06129=1095.254,-112.266,451.670,175.135,14.768,152.155
C06130=1095.260,-112.016,451.661,175.136,14.768,152.155
C06131=1095.266,-111.767,451.651,175.138,14.769,152.155
C06132=1095.273,-111.517,451.641,175.140,14.769,152.154
C06133=1095.279,-111.268,451.631,175.141,14.769,152.154
C06134=1095.284,-111.017,451.621,175.143,14.770,152.154
C06135=1095.290,-110.768,451.611,175.144,14.770,152.153
C06136=1095.297,-110.518,451.602,175.146,14.770,152.153
C06137=1095.303,-110.268,451.592,175.147,14.770,152.153
C06138=1095.309,-110.018,451.583,175.149,14.771,152.152
C06139=1095.315,-109.768,451.573,175.151,14.771,152.152
C06140=1095.321,-109.519,451.564,175.152,14.772,152.152
C06141=1095.328,-109.269,451.553,175.155,14.772,152.151
C06142=1095.334,-109.020,451.544,175.156,14.772,152.151
C06143=1095.340,-108.770,451.534,175.158,14.773,152.151
C06144=1095.346,-108.520,451.525,175.160,14.773,152.151
C06145=1095.352,-108.270,451.514,175.161,14.773,152.150
C06146=1095.358,-108.020,451.505,175.163,14.774,152.150
C06147=1095.364,-107.771,451.495,175.164,14.773,152.150
C06148=1095.371,-107.521,451.485,175.166,14.774,152.149
C06149=1095.377,-107.271,451.475,175.168,14.775,152.149
C06150=1095.383,-107.022,451.466,175.169,14.774,152.149
C06151=1095.388,-106.771,451.456,175.171,14.775,152.148
C06152=1095.394,-106.522,451.446,175.172,14.775,152.148
C06153=1095.401,-106.273,451.436,175.174,14.776,152.148
C06154=1095.407,-106.023,451.426,175.177,14.776,152.148
C06155=1095.413,-105.773,451.417,175.178,14.776,152.147
C06156=1095.419,-105.523,451.407,175.180,14.777,152.147
C06157=1095.425,-105.274,451.396,175.181,14.777,152.147
C06158=1095.431,-105.024,451.387,175.183,14.777,152.146
C06159=1095.438,-104.774,451.377,175.185,14.778,152.146
C06160=1095.443,-104.524,451.367,175.186,14.778,152.146
C06161=1095.449,-104.274,451.357,175.188,14.779,152.146
C06162=1095.456,-104.025,451.347,175.189,14.778,152.145
C06163=1095.462,-103.775,451.338,175.191,14.779,152.145
C06164=1095.467,-103.525,451.327,175.193,14.780,152.145
C06165=1095.474,-103.276,451.317,175.194,14.780,152.144
C06166=1095.480,-103.026,451.308,175.196,14.780,152.144
C06167=1095.486,-102.776,451.298,175.198,14.781,152.144
C06168=1095.491,-102.526,451.288,175.199,14.781,152.144
C06169=1095.498,-102.277,451.278,175.201,14.782,152.143
C06170=1095.504,-102.027,451.268,175.203,14.782,152.143
C06171=1095.510,-101.777,451.258,175.204,14.782,152.143
C06172=1095.516,-101.528,451.248,175.206,14.783,152.142
C06173=1095.522,-101.278,451.238,175.207,14.783,152.142
C06174=1095.528,-101.028,451.228,175.209,14.783,152.142
C06175=1095.534,-100.779,451.217,175.211,14.784,152.141
C06176=1095.540,-100.529,451.208,175.213,14.784,152.141
C06177=1095.546,-100.279,451.198,175.214,14.784,152.141
C06178=1095.553,-100.030,451.188,175.216,14.785,152.141
C06179=1095.558,-99.780,451.178,175.217,14.785,152.140
C06180=1095.565,-99.530,451.168,175.220,14.785,152.140
C06181=1095.571,-99.281,451.158,175.222,14.786,152.140
C06182=1095.576,-99.031,451.148,175.223,14.786,152.140
C06183=1095.583,-98.780,451.138,175.225,14.787,152.139
C06184=1095.590,-98.531,451.128,175.227,14.787,152.139
C06185=1095.595,-98.281,451.118,175.228,14.787,152.139
C06186=1095.602,-98.032,451.107,175.230,14.788,152.138
C06187=1095.608,-97.782,451.098,175.231,14.788,152.138
C06188=1095.613,-97.532,451.088,175.233,14.789,152.138
C06189=1095.620,-97.283,451.077,175.235,14.790,152.138
C06190=1095.626,-97.009,451.066,175.237,14.790,152.137
C06191=1095.632,-96.735,451.055,175.238,14.790,152.137
C06192=1095.639,-96.461,451.044,175.240,14.791,152.137
C06193=1095.646,-96.187,451.033,175.242,14.791,152.136
C06194=1095.652,-95.937,451.022,175.244,14.791,152.136
C06195=1095.658,-95.687,451.013,175.245,14.792,152.136
C06196=1095.664,-95.438,451.002,175.247,14.792,152.135
C06197=1095.670,-95.188,450.992,175.249,14.793,152.135
C06198=1095.675,-94.939,450.981,175.251,14.794,152.135
C06199=1095.682,-94.689,450.972,175.252,14.794,152.135
C06200=1095.687,-94.439,450.961,175.254,14.795,152.134
C06201=1095.694,-94.190,450.951,175.256,14.795,152.134
C06202=1095.699,-93.940,450.941,175.257,14.795,152.134
C06203=1095.705,-93.690,450.931,175.259,14.796,152.133
C06204=1095.711,-93.440,450.921,175.261,14.796,152.133
C06205=1095.718,-93.190,450.910,175.262,14.796,152.133
C06206=1095.723,-92.940,450.900,175.264,14.797,152.133
C06207=1095.730,-92.691,450.890,175.266,14.798,152.132
C06208=1095.735,-92.441,450.879,175.267,14.798,152.132
C06209=1095.742,-92.192,450.869,175.269,14.799,152.132
C06210=1095.747,-91.942,450.859,175.271,14.799,152.132
C06211=1095.754,-91.693,450.849,175.272,14.799,152.131
C06212=1095.759,-91.443,450.838,175.274,14.800,152.131
C06213=1095.766,-91.193,450.828,175.276,14.800,152.131
C06214=1095.772,-90.943,450.817,175.278,14.801,152.131
C06215=1095.778,-90.693,450.807,175.279,14.801,152.130
C06216=1095.784,-90.444,450.796,175.281,14.802,152.130
C06217=1095.789,-90.194,450.786,175.283,14.803,152.130
C06218=1095.796,-89.944,450.776,175.284,14.803,152.130
C06219=1095.802,-89.695,450.765,175.286,14.804,152.129
C06220=1095.808,-89.445,450.756,175.287,14.804,152.129
C06221=1095.813,-89.196,450.745,175.290,14.804,152.129
C06222=1095.820,-88.945,450.735,175.291,14.805,152.128
C06223=1095.826,-88.696,450.724,175.293,14.805,152.128
C06224=1095.832,-88.447,450.714,175.294,14.806,152.128
C06225=1095.838,-88.196,450.703,175.296,14.806,152.128
C06226=1095.844,-87.947,450.693,175.297,14.807,152.127
C06227=1095.850,-87.697,450.683,175.299,14.808,152.127
C06228=1095.856,-87.447,450.672,175.301,14.808,152.127
C06229=1095.863,-87.198,450.661,175.302,14.808,152.127
C06230=1095.868,-86.948,450.651,175.304,14.809,152.126
C06231=1095.874,-86.698,450.640,175.306,14.809,152.126
C06232=1095.880,-86.449,450.630,175.308,14.809,152.126
C06233=1095.886,-86.198,450.620,175.309,14.810,152.125
C06234=1095.893,-85.949,450.609,175.311,14.811,152.125
C06235=1095.898,-85.699,450.598,175.313,14.812,152.125
C06236=1095.904,-85.449,450.588,175.314,14.812,152.125
C06237=1095.910,-85.200,450.578,175.316,14.812,152.124
C06238=1095.917,-84.950,450.567,175.318,14.813,152.124
C06239=1095.923,-84.701,450.557,175.320,14.814,152.124
C06240=1095.929,-84.451,450.546,175.321,14.814,152.124
C06241=1095.934,-84.201,450.535,175.323,14.815,152.123
C06242=1095.941,-83.951,450.525,175.325,14.815,152.123
C06243=1095.947,-83.702,450.514,175.327,14.816,152.123
C06244=1095.953,-83.452,450.504,175.328,14.816,152.122
C06245=1095.959,-83.203,450.494,175.330,14.816,152.122
C06246=1095.965,-82.953,450.483,175.332,14.817,152.122
C06247=1095.972,-82.703,450.472,175.334,14.818,152.122
C06248=1095.977,-82.453,450.462,175.335,14.818,152.121
C06249=1095.983,-82.204,450.451,175.337,14.819,152.121
C06250=1095.990,-81.954,450.441,175.339,14.819,152.121
C06251=1095.996,-81.704,450.429,175.341,14.820,152.121
C06252=1096.001,-81.454,450.419,175.342,14.820,152.120
C06253=1096.008,-81.205,450.409,175.344,14.821,152.120
C06254=1096.015,-80.933,450.397,175.346,14.821,152.120
C06255=1096.021,-80.662,450.385,175.348,14.822,152.119
C06256=1096.028,-80.390,450.374,175.350,14.823,152.119
C06257=1096.034,-80.119,450.362,175.351,14.823,152.119
C06258=1096.041,-79.869,450.351,175.353,14.823,152.119
C06259=1096.046,-79.619,450.340,175.354,14.824,152.118
C06260=1096.052,-79.369,450.330,175.356,14.825,152.118
C06261=1096.058,-79.120,450.320,175.358,14.826,152.118
C06262=1096.065,-78.870,450.309,175.360,14.826,152.118
C06263=1096.070,-78.620,450.298,175.361,14.826,152.117
C06264=1096.076,-78.371,450.287,175.363,14.827,152.117
C06265=1096.082,-78.121,450.276,175.365,14.828,152.117
C06266=1096.088,-77.871,450.265,175.367,14.829,152.117
C06267=1096.094,-77.621,450.255,175.368,14.829,152.116
C06268=1096.100,-77.372,450.244,175.370,14.829,152.116
C06269=1096.106,-77.122,450.233,175.372,14.830,152.116
C06270=1096.112,-76.872,450.222,175.374,14.831,152.116
C06271=1096.118,-76.623,450.211,175.375,14.831,152.115
C06272=1096.124,-76.373,450.200,175.377,14.832,152.115
C06273=1096.130,-76.124,450.190,175.378,14.832,152.115
C06274=1096.137,-75.874,450.179,175.380,14.833,152.115
C06275=1096.142,-75.624,450.168,175.382,14.834,152.114
C06276=1096.148,-75.375,450.157,175.384,14.834,152.114
C06277=1096.154,-75.125,450.146,175.385,14.835,152.114
C06278=1096.160,-74.874,450.136,175.387,14.835,152.113
C06279=1096.166,-74.625,450.125,175.389,14.836,152.113
C06280=1096.172,-74.376,450.115,175.391,14.837,152.113
C06281=1096.178,-74.126,450.103,175.392,14.837,152.113
C06282=1096.184,-73.876,450.092,175.394,14.838,152.112
C06283=1096.190,-73.627,450.082,175.396,14.838,152.112
C06284=1096.196,-73.377,450.071,175.398,14.839,152.112
C06285=1096.202,-73.127,450.059,175.400,14.840,152.112
C06286=1096.208,-72.877,450.049,175.401,14.840,152.111
C06287=1096.213,-72.628,450.038,175.402,14.841,152.111
C06288=1096.218,-72.378,450.026,175.404,14.842,152.111
C06289=1096.225,-72.128,450.015,175.406,14.842,152.111
C06290=1096.230,-71.878,450.004,175.408,14.843,152.111
C06291=1096.236,-71.629,449.993,175.410,14.844,152.110
C06292=1096.243,-71.379,449.982,175.411,14.844,152.110
C06293=1096.248,-71.129,449.971,175.413,14.845,152.110
C06294=1096.254,-70.880,449.960,175.415,14.845,152.110
C06295=1096.260,-70.630,449.949,175.417,14.846,152.109
C06296=1096.266,-70.380,449.938,175.418,14.847,152.109
C06297=1096.272,-70.131,449.927,175.420,14.848,152.109
C06298=1096.278,-69.881,449.916,175.421,14.848,152.109
C06299=1096.284,-69.632,449.904,175.423,14.849,152.108
C06300=1096.290,-69.382,449.893,175.425,14.850,152.108
C06301=1096.296,-69.133,449.883,175.427,14.850,152.108
C06302=1096.301,-68.883,449.872,175.429,14.851,152.108
C06303=1096.308,-68.633,449.860,175.430,14.852,152.107
C06304=1096.313,-68.383,449.849,175.432,14.852,152.107
C06305=1096.319,-68.134,449.838,175.433,14.853,152.107
C06306=1096.325,-67.883,449.827,175.435,14.853,152.107
C06307=1096.331,-67.634,449.816,175.437,14.854,152.106
C06308=1096.336,-67.384,449.805,175.439,14.855,152.106
C06309=1096.343,-67.135,449.793,175.441,14.856,152.106
C06310=1096.349,-66.885,449.782,175.443,14.857,152.106
C06311=1096.354,-66.636,449.771,175.444,14.857,152.106
C06312=1096.361,-66.386,449.760,175.446,14.858,152.105
C06313=1096.367,-66.136,449.749,175.447,14.858,152.105
C06314=1096.372,-65.886,449.737,175.449,14.859,152.105
C06315=1096.378,-65.637,449.726,175.451,14.860,152.104
C06316=1096.384,-65.387,449.715,175.453,14.860,152.104
C06317=1096.390,-65.137,449.704,175.455,14.861,152.104
C06318=1096.396,-64.868,449.691,175.457,14.862,152.104
C06319=1096.403,-64.598,449.680,175.459,14.863,152.103
C06320=1096.409,-64.329,449.667,175.461,14.863,152.103
C06321=1096.416,-64.059,449.656,175.463,14.864,152.103
C06322=1096.422,-63.811,449.644,175.464,14.864,152.103
C06323=1096.428,-63.560,449.633,175.466,14.865,152.102
C06324=1096.433,-63.311,449.621,175.467,14.866,152.102
C06325=1096.439,-63.061,449.610,175.469,14.867,152.102
C06326=1096.446,-62.812,449.599,175.471,14.868,152.102
C06327=1096.451,-62.562,449.588,175.473,14.868,152.101
C06328=1096.458,-62.312,449.576,175.475,14.869,152.101
C06329=1096.463,-62.062,449.566,175.476,14.869,152.101
C06330=1096.469,-61.813,449.553,175.478,14.870,152.101
C06331=1096.475,-61.563,449.542,175.479,14.871,152.100
C06332=1096.481,-61.313,449.531,175.481,14.871,152.100
C06333=1096.487,-61.064,449.519,175.483,14.872,152.100
C06334=1096.493,-60.814,449.508,175.485,14.873,152.100
C06335=1096.500,-60.564,449.497,175.487,14.873,152.099
C06336=1096.505,-60.314,449.486,175.489,14.875,152.099
C06337=1096.511,-60.065,449.474,175.490,14.875,152.099
C06338=1096.517,-59.815,449.463,175.492,14.875,152.099
C06339=1096.523,-59.566,449.452,175.493,14.876,152.099
C06340=1096.529,-59.316,449.440,175.495,14.877,152.098
C06341=1096.534,-59.066,449.429,175.497,14.878,152.098
C06342=1096.541,-58.816,449.417,175.499,14.878,152.098
C06343=1096.547,-58.567,449.406,175.501,14.879,152.098
C06344=1096.553,-58.317,449.394,175.503,14.880,152.097
C06345=1096.559,-58.068,449.383,175.505,14.881,152.097
C06346=1096.565,-57.818,449.371,175.506,14.881,152.097
C06347=1096.570,-57.568,449.360,175.508,14.881,152.096
C06348=1096.577,-57.319,449.348,175.509,14.883,152.096
C06349=1096.583,-57.069,449.337,175.511,14.883,152.096
C06350=1096.589,-56.819,449.325,175.513,14.884,152.096
C06351=1096.594,-56.570,449.314,175.515,14.885,152.096
C06352=1096.601,-56.320,449.303,175.517,14.885,152.095
C06353=1096.607,-56.071,449.291,175.519,14.886,152.095
C06354=1096.612,-55.820,449.279,175.521,14.887,152.095
C06355=1096.618,-55.572,449.268,175.522,14.888,152.095
C06356=1096.625,-55.321,449.256,175.524,14.888,152.094
C06357=1096.631,-55.072,449.244,175.525,14.888,152.094
C06358=1096.636,-54.822,449.233,175.527,14.889,152.094
C06359=1096.643,-54.572,449.221,175.529,14.890,152.094
C06360=1096.649,-54.323,449.210,175.531,14.891,152.093
C06361=1096.656,-54.073,449.198,175.533,14.891,152.093
C06362=1096.661,-53.824,449.187,175.535,14.893,152.093
C06363=1096.667,-53.574,449.175,175.536,14.893,152.093
C06364=1096.673,-53.324,449.164,175.538,14.894,152.092
C06365=1096.679,-53.075,449.151,175.540,14.895,152.092
C06366=1096.685,-52.824,449.140,175.542,14.895,152.092
C06367=1096.691,-52.576,449.128,175.543,14.896,152.092
C06368=1096.698,-52.325,449.117,175.545,14.896,152.091
C06369=1096.703,-52.076,449.105,175.547,14.897,152.091
C06370=1096.709,-51.826,449.094,175.549,14.898,152.091
C06371=1096.715,-51.577,449.082,175.551,14.898,152.091
C06372=1096.721,-51.327,449.070,175.553,14.899,152.090
C06373=1096.727,-51.077,449.058,175.555,14.900,152.090
C06374=1096.734,-50.828,449.047,175.556,14.901,152.090
C06375=1096.739,-50.578,449.035,175.558,14.901,152.090
C06376=1096.745,-50.329,449.023,175.560,14.903,152.089
C06377=1096.751,-50.078,449.012,175.562,14.903,152.089
C06378=1096.757,-49.829,449.000,175.564,14.904,152.089
C06379=1096.763,-49.579,448.987,175.565,14.905,152.089
C06380=1096.768,-49.330,448.976,175.567,14.905,152.088
C06381=1096.774,-49.080,448.964,175.569,14.906,152.088
C06382=1096.781,-48.812,448.952,175.571,14.907,152.088
C06383=1096.787,-48.544,448.939,175.573,14.908,152.088
C06384=1096.794,-48.276,448.926,175.575,14.909,152.088
C06385=1096.800,-48.008,448.913,175.576,14.910,152.087
C06386=1096.806,-47.758,448.901,175.578,14.910,152.087
C06387=1096.811,-47.508,448.890,175.580,14.911,152.087
C06388=1096.818,-47.259,448.878,175.582,14.912,152.086
C06389=1096.823,-47.010,448.866,175.584,14.912,152.086
C06390=1096.829,-46.759,448.854,175.586,14.913,152.086
C06391=1096.835,-46.510,448.842,175.587,14.914,152.086
C06392=1096.841,-46.260,448.830,175.589,14.915,152.086
C06393=1096.847,-46.011,448.819,175.591,14.916,152.085
C06394=1096.852,-45.761,448.806,175.593,14.917,152.085
C06395=1096.859,-45.511,448.794,175.594,14.917,152.085
C06396=1096.864,-45.262,448.783,175.596,14.917,152.085
C06397=1096.870,-45.012,448.770,175.598,14.919,152.084
C06398=1096.876,-44.763,448.759,175.600,14.919,152.084
C06399=1096.882,-44.513,448.746,175.601,14.920,152.084
C06400=1096.888,-44.263,448.735,175.603,14.921,152.084
C06401=1096.894,-44.014,448.723,175.605,14.922,152.083
C06402=1096.900,-43.764,448.711,175.607,14.922,152.083
C06403=1096.906,-43.514,448.698,175.609,14.923,152.083
C06404=1096.911,-43.264,448.687,175.611,14.924,152.083
C06405=1096.918,-43.015,448.675,175.612,14.925,152.083
C06406=1096.923,-42.766,448.663,175.614,14.926,152.082
C06407=1096.930,-42.516,448.651,175.616,14.926,152.082
C06408=1096.936,-42.266,448.638,175.618,14.927,152.082
C06409=1096.941,-42.016,448.627,175.620,14.928,152.081
C06410=1096.947,-41.767,448.615,175.622,14.929,152.081
C06411=1096.953,-41.517,448.602,175.624,14.929,152.081
C06412=1096.959,-41.268,448.590,175.626,14.930,152.081
C06413=1096.965,-41.018,448.578,175.627,14.931,152.081
C06414=1096.971,-40.768,448.566,175.629,14.932,152.080
C06415=1096.977,-40.519,448.555,175.631,14.933,152.080
C06416=1096.983,-40.269,448.542,175.633,14.933,152.080
C06417=1096.989,-40.019,448.530,175.635,14.934,152.080
C06418=1096.995,-39.770,448.518,175.637,14.935,152.079
C06419=1097.001,-39.520,448.505,175.638,14.936,152.079
C06420=1097.007,-39.270,448.493,175.640,14.936,152.079
C06421=1097.013,-39.021,448.481,175.642,14.938,152.079
C06422=1097.018,-38.771,448.469,175.644,14.938,152.078
C06423=1097.024,-38.521,448.457,175.646,14.939,152.078
C06424=1097.029,-38.272,448.445,175.648,14.940,152.078
C06425=1097.036,-38.022,448.433,175.649,14.940,152.078
C06426=1097.042,-37.772,448.420,175.651,14.941,152.077
C06427=1097.047,-37.523,448.408,175.653,14.942,152.077
C06428=1097.053,-37.273,448.395,175.655,14.943,152.077
C06429=1097.059,-37.023,448.383,175.657,14.944,152.077
C06430=1097.065,-36.775,448.371,175.659,14.945,152.076
C06431=1097.071,-36.525,448.359,175.660,14.945,152.076
C06432=1097.077,-36.275,448.346,175.662,14.946,152.076
C06433=1097.082,-36.026,448.334,175.664,14.947,152.076
C06434=1097.088,-35.776,448.321,175.666,14.948,152.076
C06435=1097.094,-35.526,448.309,175.668,14.949,152.075
C06436=1097.100,-35.276,448.298,175.669,14.949,152.075
C06437=1097.106,-35.026,448.285,175.671,14.950,152.075
C06438=1097.112,-34.777,448.273,175.673,14.951,152.075
C06439=1097.118,-34.527,448.260,175.675,14.952,152.074
C06440=1097.123,-34.278,448.248,175.677,14.953,152.074
C06441=1097.129,-34.028,448.235,175.679,14.954,152.074
C06442=1097.136,-33.779,448.223,175.680,14.954,152.074
C06443=1097.142,-33.529,448.210,175.682,14.955,152.073
C06444=1097.147,-33.280,448.198,175.684,14.956,152.073
C06445=1097.153,-33.030,448.186,175.686,14.956,152.073
C06446=1097.159,-32.762,448.173,175.688,14.957,152.073
C06447=1097.165,-32.494,448.159,175.691,14.958,152.072
C06448=1097.172,-32.226,448.146,175.692,14.960,152.072
C06449=1097.178,-31.959,448.132,175.694,14.960,152.072
C06450=1097.184,-31.709,448.120,175.696,14.961,152.072
C06451=1097.189,-31.460,448.108,175.698,14.962,152.071
C06452=1097.195,-31.210,448.095,175.700,14.963,152.071
C06453=1097.201,-30.960,448.082,175.702,14.963,152.071
C06454=1097.207,-30.710,448.070,175.703,14.964,152.071
C06455=1097.213,-30.461,448.058,175.705,14.965,152.070
C06456=1097.219,-30.211,448.046,175.707,14.966,152.070
C06457=1097.225,-29.961,448.033,175.709,14.967,152.070
C06458=1097.231,-29.712,448.020,175.711,14.967,152.070
C06459=1097.237,-29.462,448.007,175.713,14.968,152.070
C06460=1097.242,-29.213,447.995,175.714,14.969,152.069
C06461=1097.248,-28.963,447.983,175.716,14.970,152.069
C06462=1097.254,-28.713,447.970,175.718,14.970,152.069
C06463=1097.260,-28.464,447.958,175.720,14.971,152.069
C06464=1097.266,-28.214,447.944,175.723,14.972,152.068
C06465=1097.272,-27.965,447.932,175.725,14.973,152.068
C06466=1097.278,-27.715,447.920,175.726,14.974,152.068
C06467=1097.284,-27.465,447.907,175.728,14.975,152.068
C06468=1097.289,-27.215,447.894,175.730,14.976,152.067
C06469=1097.296,-26.966,447.882,175.732,14.977,152.067
C06470=1097.302,-26.716,447.869,175.734,14.977,152.067
C06471=1097.307,-26.467,447.856,175.736,14.978,152.067
C06472=1097.313,-26.217,447.844,175.738,14.979,152.066
C06473=1097.319,-25.968,447.831,175.739,14.980,152.066
C06474=1097.325,-25.718,447.818,175.741,14.981,152.066
C06475=1097.331,-25.468,447.805,175.743,14.981,152.066
C06476=1097.336,-25.219,447.793,175.745,14.982,152.065
C06477=1097.342,-24.970,447.780,175.747,14.983,152.065
C06478=1097.348,-24.720,447.767,175.748,14.984,152.065
C06479=1097.354,-24.470,447.755,175.750,14.984,152.065
C06480=1097.360,-24.220,447.742,175.752,14.986,152.065
C06481=1097.365,-23.971,447.729,175.755,14.987,152.064
C06482=1097.371,-23.721,447.716,175.756,14.988,152.064
C06483=1097.377,-23.471,447.704,175.758,14.988,152.064
C06484=1097.383,-23.222,447.690,175.760,14.989,152.063
C06485=1097.389,-22.972,447.678,175.762,14.990,152.063
C06486=1097.395,-22.722,447.665,175.764,14.991,152.063
C06487=1097.400,-22.474,447.652,175.766,14.991,152.063
C06488=1097.406,-22.224,447.640,175.767,14.993,152.063
C06489=1097.411,-21.974,447.627,175.769,14.993,152.062
C06490=1097.418,-21.725,447.613,175.771,14.994,152.062
C06491=1097.424,-21.475,447.601,175.773,14.995,152.062
C06492=1097.430,-21.225,447.588,175.775,14.995,152.062
C06493=1097.436,-20.975,447.575,175.777,14.996,152.061
C06494=1097.441,-20.726,447.563,175.780,14.997,152.061
C06495=1097.447,-20.477,447.549,175.781,14.998,152.061
C06496=1097.452,-20.227,447.536,175.783,14.999,152.060
C06497=1097.459,-19.978,447.523,175.785,15.000,152.060
C06498=1097.465,-19.728,447.511,175.787,15.001,152.060
C06499=1097.470,-19.478,447.498,175.789,15.002,152.060
C06500=1097.477,-19.229,447.485,175.790,15.002,152.060
C06501=1097.482,-18.978,447.472,175.792,15.003,152.059
C06502=1097.488,-18.729,447.458,175.794,15.004,152.059
C06503=1097.494,-18.479,447.446,175.796,15.005,152.059
C06504=1097.500,-18.231,447.433,175.798,15.005,152.059
C06505=1097.505,-17.981,447.420,175.801,15.007,152.058
C06506=1097.511,-17.731,447.407,175.803,15.007,152.058
C06507=1097.517,-17.481,447.394,175.804,15.008,152.058
C06508=1097.523,-17.232,447.381,175.806,15.009,152.058
C06509=1097.529,-16.982,447.368,175.808,15.010,152.057
C06510=1097.535,-16.714,447.353,175.810,15.011,152.057
C06511=1097.542,-16.445,447.340,175.812,15.012,152.057
C06512=1097.548,-16.177,447.325,175.814,15.013,152.057
C06513=1097.554,-15.908,447.312,175.816,15.014,152.056
C06514=1097.560,-15.659,447.299,175.818,15.014,152.056
C06515=1097.566,-15.409,447.286,175.820,15.015,152.056
C06516=1097.572,-15.159,447.272,175.822,15.016,152.056
C06517=1097.578,-14.910,447.260,175.824,15.017,152.055
C06518=1097.584,-14.660,447.246,175.826,15.017,152.055
C06519=1097.589,-14.410,447.233,175.828,15.019,152.055
C06520=1097.595,-14.161,447.220,175.830,15.019,152.054
C06521=1097.601,-13.911,447.206,175.832,15.020,152.054
C06522=1097.607,-13.661,447.194,175.834,15.021,152.054
C06523=1097.613,-13.412,447.180,175.836,15.022,152.054
C06524=1097.618,-13.162,447.167,175.838,15.022,152.053
C06525=1097.624,-12.913,447.154,175.839,15.023,152.053
C06526=1097.630,-12.663,447.140,175.841,15.024,152.053
C06527=1097.636,-12.413,447.128,175.844,15.026,152.053
C06528=1097.642,-12.164,447.114,175.846,15.026,152.053
C06529=1097.647,-11.914,447.100,175.847,15.027,152.052
C06530=1097.653,-11.664,447.088,175.849,15.028,152.052
C06531=1097.659,-11.415,447.074,175.851,15.028,152.052
C06532=1097.665,-11.166,447.061,175.853,15.029,152.052
C06533=1097.671,-10.916,447.048,175.855,15.030,152.051
C06534=1097.676,-10.667,447.035,175.857,15.031,152.051
C06535=1097.682,-10.418,447.021,175.860,15.032,152.051
C06536=1097.687,-10.167,447.008,175.861,15.033,152.050
C06537=1097.693,-9.918,446.995,175.863,15.033,152.050
C06538=1097.699,-9.669,446.981,175.865,15.034,152.050
C06539=1097.705,-9.418,446.968,175.867,15.035,152.050
C06540=1097.711,-9.169,446.955,175.869,15.036,152.050
C06541=1097.717,-8.919,446.941,175.871,15.037,152.049
C06542=1097.723,-8.670,446.928,175.872,15.038,152.049
C06543=1097.728,-8.420,446.915,175.875,15.039,152.049
C06544=1097.734,-8.170,446.901,175.877,15.040,152.049
C06545=1097.740,-7.921,446.888,175.879,15.040,152.048
C06546=1097.746,-7.672,446.874,175.881,15.041,152.048
C06547=1097.751,-7.421,446.861,175.883,15.042,152.048
C06548=1097.758,-7.172,446.848,175.884,15.043,152.048
C06549=1097.763,-6.923,446.834,175.886,15.043,152.047
C06550=1097.769,-6.673,446.821,175.889,15.045,152.047
C06551=1097.775,-6.424,446.807,175.891,15.045,152.047
C06552=1097.781,-6.174,446.794,175.893,15.046,152.046
C06553=1097.786,-5.924,446.780,175.895,15.047,152.046
C06554=1097.792,-5.675,446.767,175.897,15.048,152.046
C06555=1097.798,-5.425,446.753,175.898,15.048,152.046
C06556=1097.804,-5.176,446.740,175.900,15.049,152.045
C06557=1097.809,-4.927,446.726,175.903,15.050,152.045
C06558=1097.816,-4.677,446.713,175.905,15.051,152.045
C06559=1097.822,-4.427,446.699,175.907,15.052,152.045
C06560=1097.828,-4.177,446.686,175.909,15.053,152.044
C06561=1097.833,-3.928,446.672,175.910,15.053,152.044
C06562=1097.839,-3.678,446.659,175.912,15.054,152.044
C06563=1097.845,-3.429,446.645,175.914,15.055,152.044
C06564=1097.851,-3.180,446.632,175.917,15.056,152.043
C06565=1097.857,-2.930,446.618,175.919,15.057,152.043
C06566=1097.862,-2.680,446.604,175.921,15.058,152.043
C06567=1097.868,-2.431,446.591,175.923,15.058,152.043
C06568=1097.874,-2.182,446.577,175.924,15.059,152.042
C06569=1097.879,-1.932,446.563,175.926,15.060,152.042
C06570=1097.885,-1.682,446.549,175.929,15.061,152.042
C06571=1097.891,-1.432,446.536,175.931,15.062,152.041
C06572=1097.897,-1.182,446.522,175.933,15.063,152.041
C06573=1097.902,-0.933,446.509,175.935,15.063,152.041
C06574=1097.908,-0.663,446.494,175.937,15.065,152.041
C06575=1097.915,-0.392,446.479,175.939,15.066,152.040
C06576=1097.921,-0.123,446.465,175.941,15.066,152.040
C06577=1097.927,0.148,446.449,175.944,15.068,152.040
C06578=1097.933,0.398,446.435,175.946,15.068,152.040
C06579=1097.938,0.647,446.422,175.947,15.069,152.039
C06580=1097.944,0.897,446.408,175.949,15.070,152.039
C06581=1097.950,1.145,446.394,175.951,15.071,152.039
C06582=1097.956,1.395,446.380,175.953,15.071,152.039
C06583=1097.961,1.645,446.366,175.956,15.073,152.038
C06584=1097.967,1.894,446.353,175.958,15.073,152.038
C06585=1097.973,2.143,446.339,175.959,15.074,152.038
C06586=1097.979,2.394,446.325,175.961,15.075,152.037
C06587=1097.984,2.643,446.311,175.963,15.076,152.037
C06588=1097.991,2.893,446.297,175.966,15.077,152.037
C06589=1097.996,3.142,446.284,175.968,15.078,152.037
C06590=1098.001,3.392,446.270,175.970,15.078,152.036
C06591=1098.007,3.641,446.256,175.971,15.079,152.036
C06592=1098.013,3.892,446.242,175.974,15.079,152.036
C06593=1098.020,4.140,446.228,175.976,15.081,152.035
C06594=1098.025,4.390,446.214,175.978,15.081,152.035
C06595=1098.030,4.639,446.200,175.980,15.082,152.035
C06596=1098.036,4.889,446.186,175.982,15.083,152.035
C06597=1098.041,5.139,446.172,175.984,15.084,152.034
C06598=1098.048,5.389,446.159,175.986,15.084,152.034
C06599=1098.054,5.638,446.145,175.988,15.086,152.034
C06600=1098.060,5.887,446.130,175.990,15.087,152.034
C06601=1098.065,6.137,446.116,175.992,15.087,152.033
C06602=1098.070,6.386,446.102,175.994,15.088,152.033
C06603=1098.077,6.636,446.088,175.996,15.089,152.033
C06604=1098.083,6.886,446.075,175.999,15.090,152.033
C06605=1098.089,7.135,446.060,176.001,15.090,152.032
C06606=1098.094,7.384,446.046,176.003,15.091,152.032
C06607=1098.100,7.635,446.032,176.005,15.092,152.032
C06608=1098.106,7.884,446.018,176.006,15.093,152.031
C06609=1098.111,8.133,446.004,176.009,15.094,152.031
C06610=1098.117,8.383,445.990,176.011,15.095,152.031
C06611=1098.124,8.633,445.976,176.013,15.095,152.031
C06612=1098.129,8.882,445.962,176.015,15.096,152.030
C06613=1098.135,9.131,445.948,176.017,15.096,152.030
C06614=1098.140,9.381,445.934,176.020,15.098,152.030
C06615=1098.146,9.631,445.920,176.021,15.098,152.029
C06616=1098.152,9.880,445.905,176.023,15.099,152.029
C06617=1098.158,10.130,445.891,176.025,15.100,152.029
C06618=1098.163,10.379,445.877,176.027,15.101,152.029
C06619=1098.170,10.629,445.862,176.030,15.102,152.028
C06620=1098.176,10.878,445.849,176.032,15.102,152.028
C06621=1098.181,11.128,445.835,176.034,15.103,152.028
C06622=1098.188,11.377,445.820,176.036,15.104,152.027
C06623=1098.193,11.627,445.807,176.038,15.105,152.027
C06624=1098.199,11.876,445.793,176.040,15.106,152.027
C06625=1098.204,12.125,445.778,176.042,15.106,152.026
C06626=1098.210,12.376,445.764,176.044,15.107,152.026
C06627=1098.216,12.625,445.749,176.046,15.108,152.026
C06628=1098.222,12.874,445.735,176.049,15.109,152.026
C06629=1098.228,13.124,445.720,176.051,15.110,152.025
C06630=1098.234,13.373,445.707,176.053,15.110,152.025
C06631=1098.239,13.623,445.693,176.055,15.111,152.025
C06632=1098.245,13.873,445.678,176.057,15.111,152.024
C06633=1098.252,14.122,445.665,176.059,15.113,152.024
C06634=1098.258,14.372,445.650,176.061,15.114,152.024
C06635=1098.263,14.621,445.635,176.063,15.114,152.023
C06636=1098.269,14.870,445.621,176.065,15.115,152.023
C06637=1098.274,15.120,445.607,176.068,15.116,152.023
C06638=1098.281,15.393,445.591,176.070,15.117,152.023
C06639=1098.287,15.664,445.575,176.072,15.117,152.022
C06640=1098.293,15.937,445.559,176.075,15.118,152.022
C06641=1098.300,16.208,445.544,176.077,15.119,152.022
C06642=1098.306,16.459,445.530,176.079,15.120,152.021
C06643=1098.312,16.707,445.515,176.081,15.121,152.021
C06644=1098.316,16.957,445.501,176.083,15.121,152.021
C06645=1098.323,17.207,445.486,176.085,15.122,152.021
C06646=1098.328,17.457,445.472,176.088,15.123,152.020
C06647=1098.334,17.706,445.457,176.090,15.124,152.020
C06648=1098.340,17.956,445.443,176.092,15.124,152.020
C06649=1098.346,18.205,445.428,176.094,15.125,152.019
C06650=1098.351,18.454,445.414,176.096,15.126,152.019
C06651=1098.357,18.704,445.399,176.098,15.127,152.019
C06652=1098.363,18.953,445.384,176.100,15.128,152.018
C06653=1098.369,19.204,445.370,176.102,15.128,152.018
C06654=1098.375,19.452,445.356,176.104,15.129,152.018
C06655=1098.380,19.702,445.342,176.107,15.130,152.018
C06656=1098.386,19.952,445.327,176.109,15.131,152.017
C06657=1098.392,20.201,445.312,176.111,15.131,152.017
C06658=1098.397,20.451,445.298,176.113,15.132,152.017
C06659=1098.403,20.700,445.283,176.115,15.133,152.016
C06660=1098.409,20.949,445.268,176.118,15.134,152.016
C06661=1098.415,21.199,445.254,176.120,15.134,152.016
C06662=1098.420,21.449,445.239,176.121,15.135,152.015
C06663=1098.426,21.698,445.224,176.124,15.137,152.015
C06664=1098.432,21.948,445.210,176.126,15.137,152.015
C06665=1098.438,22.197,445.195,176.128,15.138,152.014
C06666=1098.444,22.447,445.180,176.130,15.138,152.014
C06667=1098.449,22.696,445.166,176.133,15.140,152.014
C06668=1098.455,22.945,445.151,176.135,15.140,152.013
C06669=1098.460,23.195,445.136,176.137,15.141,152.013
C06670=1098.466,23.444,445.121,176.139,15.141,152.013
C06671=1098.472,23.695,445.107,176.142,15.142,152.013
C06672=1098.478,23.944,445.092,176.143,15.143,152.012
C06673=1098.484,24.194,445.077,176.145,15.144,152.012
C06674=1098.489,24.442,445.062,176.148,15.145,152.012
C06675=1098.495,24.692,445.048,176.150,15.145,152.011
C06676=1098.501,24.942,445.033,176.152,15.146,152.011
C06677=1098.506,25.191,445.018,176.154,15.146,152.011
C06678=1098.513,25.441,445.003,176.157,15.148,152.010
C06679=1098.518,25.690,444.988,176.159,15.149,152.010
C06680=1098.524,25.940,444.974,176.161,15.149,152.010
C06681=1098.530,26.189,444.959,176.163,15.150,152.009
C06682=1098.536,26.439,444.944,176.166,15.151,152.009
C06683=1098.541,26.688,444.929,176.168,15.151,152.009
C06684=1098.547,26.938,444.914,176.170,15.152,152.008
C06685=1098.553,27.187,444.899,176.171,15.153,152.008
C06686=1098.559,27.437,444.884,176.174,15.154,152.008
C06687=1098.564,27.686,444.870,176.176,15.154,152.008
C06688=1098.570,27.936,444.855,176.179,15.155,152.007
C06689=1098.576,28.185,444.840,176.181,15.156,152.007
C06690=1098.582,28.435,444.825,176.183,15.157,152.007
C06691=1098.587,28.684,444.810,176.185,15.157,152.006
C06692=1098.594,28.934,444.795,176.187,15.158,152.006
C06693=1098.599,29.183,444.780,176.190,15.159,152.006
C06694=1098.604,29.432,444.765,176.192,15.159,152.005
C06695=1098.610,29.682,444.750,176.194,15.160,152.005
C06696=1098.616,29.931,444.735,176.197,15.161,152.004
C06697=1098.622,30.181,444.720,176.199,15.162,152.004
C06698=1098.627,30.430,444.705,176.201,15.162,152.004
C06699=1098.633,30.680,444.690,176.203,15.163,152.004
C06700=1098.639,30.929,444.675,176.205,15.164,152.003
C06701=1098.644,31.179,444.660,176.208,15.164,152.003
C06702=1098.651,31.452,444.643,176.210,15.166,152.003
C06703=1098.657,31.726,444.627,176.212,15.166,152.002
C06704=1098.664,32.000,444.610,176.215,15.167,152.002
C06705=1098.669,32.273,444.594,176.217,15.168,152.001
C06706=1098.675,32.523,444.578,176.219,15.168,152.001
C06707=1098.681,32.772,444.564,176.222,15.169,152.001
C06708=1098.687,33.022,444.548,176.224,15.170,152.001
C06709=1098.692,33.271,444.534,176.226,15.170,152.000
C06710=1098.698,33.521,444.518,176.229,15.172,152.000
C06711=1098.704,33.770,444.504,176.231,15.172,152.000
C06712=1098.709,34.020,444.488,176.233,15.173,151.999
C06713=1098.716,34.269,444.473,176.235,15.173,151.999
C06714=1098.721,34.519,444.458,176.238,15.174,151.998
C06715=1098.728,34.768,444.442,176.240,15.175,151.998
C06716=1098.733,35.017,444.427,176.242,15.175,151.998
C06717=1098.738,35.267,444.412,176.245,15.177,151.997
C06718=1098.745,35.517,444.397,176.247,15.177,151.997
C06719=1098.750,35.766,444.381,176.249,15.178,151.997
C06720=1098.756,36.016,444.366,176.252,15.178,151.996
C06721=1098.761,36.265,444.351,176.253,15.179,151.996
C06722=1098.768,36.514,444.336,176.256,15.179,151.996
C06723=1098.773,36.764,444.320,176.257,15.180,151.995
C06724=1098.778,37.013,444.305,176.260,15.181,151.995
C06725=1098.785,37.263,444.290,176.263,15.181,151.995
C06726=1098.790,37.512,444.275,176.265,15.182,151.994
C06727=1098.796,37.762,444.260,176.267,15.183,151.994
C06728=1098.802,38.011,444.244,176.269,15.184,151.994
C06729=1098.807,38.260,444.228,176.272,15.184,151.993
C06730=1098.813,38.510,444.213,176.274,15.185,151.993
C06731=1098.819,38.760,444.198,176.276,15.186,151.993
C06732=1098.825,39.009,444.182,176.278,15.186,151.992
C06733=1098.830,39.259,444.166,176.281,15.187,151.992
C06734=1098.836,39.507,444.152,176.283,15.188,151.992
C06735=1098.842,39.757,444.136,176.285,15.188,151.991
C06736=1098.848,40.007,444.120,176.288,15.190,151.991
C06737=1098.853,40.256,444.105,176.290,15.190,151.990
C06738=1098.859,40.506,444.090,176.292,15.190,151.990
C06739=1098.864,40.754,444.074,176.295,15.192,151.990
C06740=1098.870,41.004,444.059,176.297,15.192,151.989
C06741=1098.876,41.254,444.043,176.299,15.193,151.989
C06742=1098.881,41.504,444.028,176.301,15.193,151.989
C06743=1098.887,41.753,444.012,176.304,15.194,151.988
C06744=1098.893,42.003,443.997,176.306,15.195,151.988
C06745=1098.898,42.252,443.981,176.308,15.195,151.988
C06746=1098.904,42.501,443.965,176.311,15.196,151.987
C06747=1098.910,42.751,443.950,176.313,15.196,151.987
C06748=1098.916,42.999,443.934,176.315,15.197,151.986
C06749=1098.921,43.249,443.919,176.318,15.198,151.986
C06750=1098.927,43.499,443.903,176.320,15.198,151.986
C06751=1098.933,43.749,443.887,176.322,15.199,151.986
C06752=1098.938,43.998,443.872,176.325,15.200,151.985
C06753=1098.944,44.247,443.856,176.327,15.200,151.985
C06754=1098.950,44.496,443.841,176.329,15.201,151.984
C06755=1098.955,44.746,443.825,176.332,15.202,151.984
C06756=1098.961,44.996,443.809,176.334,15.203,151.984
C06757=1098.966,45.245,443.794,176.337,15.204,151.983
C06758=1098.972,45.494,443.778,176.339,15.204,151.983
C06759=1098.978,45.744,443.762,176.341,15.205,151.983
C06760=1098.983,45.993,443.746,176.344,15.205,151.982
C06761=1098.989,46.243,443.731,176.346,15.206,151.982
C06762=1098.995,46.492,443.715,176.348,15.207,151.982
C06763=1099.000,46.741,443.699,176.351,15.207,151.981
C06764=1099.006,46.991,443.683,176.353,15.208,151.981
C06765=1099.012,47.241,443.668,176.355,15.208,151.980
C06766=1099.018,47.514,443.650,176.358,15.209,151.980
C06767=1099.024,47.788,443.633,176.360,15.210,151.980
C06768=1099.030,48.061,443.615,176.363,15.210,151.979
C06769=1099.036,48.335,443.598,176.366,15.212,151.979
C06770=1099.042,48.585,443.582,176.368,15.212,151.978
C06771=1099.048,48.834,443.566,176.370,15.212,151.978
C06772=1099.053,49.083,443.551,176.373,15.213,151.978
C06773=1099.059,49.333,443.534,176.375,15.214,151.977
C06774=1099.064,49.583,443.519,176.377,15.214,151.977
C06775=1099.070,49.832,443.503,176.380,15.215,151.976
C06776=1099.076,50.081,443.487,176.382,15.216,151.976
C06777=1099.081,50.331,443.471,176.384,15.216,151.976
C06778=1099.087,50.580,443.455,176.387,15.217,151.975
C06779=1099.093,50.829,443.439,176.389,15.217,151.975
C06780=1099.098,51.079,443.424,176.392,15.219,151.975
C06781=1099.104,51.328,443.407,176.394,15.219,151.974
C06782=1099.110,51.577,443.391,176.396,15.219,151.974
C06783=1099.116,51.827,443.375,176.399,15.220,151.973
C06784=1099.122,52.077,443.359,176.402,15.221,151.973
C06785=1099.127,52.325,443.343,176.403,15.221,151.973
C06786=1099.133,52.575,443.328,176.406,15.222,151.972
C06787=1099.139,52.825,443.312,176.409,15.222,151.972
C06788=1099.144,53.074,443.295,176.411,15.223,151.971
C06789=1099.150,53.324,443.279,176.414,15.224,151.971
C06790=1099.155,53.573,443.263,176.416,15.224,151.971
C06791=1099.161,53.822,443.247,176.418,15.225,151.970
C06792=1099.167,54.072,443.231,176.421,15.226,151.970
C06793=1099.172,54.322,443.215,176.423,15.226,151.969
C06794=1099.178,54.571,443.199,176.426,15.227,151.969
C06795=1099.184,54.820,443.183,176.428,15.227,151.969
C06796=1099.190,55.070,443.166,176.430,15.227,151.968
C06797=1099.196,55.318,443.151,176.433,15.229,151.968
C06798=1099.201,55.569,443.134,176.435,15.229,151.968
C06799=1099.206,55.818,443.118,176.437,15.229,151.967
C06800=1099.212,56.067,443.102,176.440,15.230,151.967
C06801=1099.218,56.317,443.086,176.442,15.230,151.966
C06802=1099.224,56.566,443.069,176.445,15.231,151.966
C06803=1099.230,56.815,443.053,176.448,15.232,151.965
C06804=1099.236,57.065,443.038,176.450,15.232,151.965
C06805=1099.241,57.315,443.021,176.453,15.233,151.965
C06806=1099.246,57.564,443.005,176.455,15.233,151.964
C06807=1099.252,57.813,442.989,176.457,15.233,151.964
C06808=1099.258,58.062,442.972,176.460,15.234,151.963
C06809=1099.264,58.312,442.956,176.462,15.235,151.963
C06810=1099.270,58.561,442.940,176.465,15.235,151.962
C06811=1099.276,58.811,442.923,176.467,15.236,151.962
C06812=1099.281,59.060,442.907,176.469,15.237,151.962
C06813=1099.287,59.309,442.890,176.472,15.237,151.961
C06814=1099.293,59.559,442.874,176.475,15.238,151.961
C06815=1099.299,59.808,442.858,176.477,15.238,151.960
C06816=1099.305,60.058,442.842,176.480,15.239,151.960
C06817=1099.310,60.308,442.826,176.482,15.239,151.959
C06818=1099.316,60.557,442.809,176.485,15.240,151.959
C06819=1099.322,60.806,442.793,176.487,15.240,151.959
C06820=1099.328,61.056,442.777,176.490,15.240,151.958
C06821=1099.333,61.305,442.760,176.492,15.241,151.958
C06822=1099.339,61.555,442.744,176.495,15.241,151.957
C06823=1099.345,61.803,442.727,176.497,15.242,151.957
C06824=1099.351,62.053,442.710,176.500,15.243,151.957
C06825=1099.357,62.302,442.694,176.502,15.243,151.956
C06826=1099.363,62.552,442.677,176.505,15.244,151.956
C06827=1099.369,62.801,442.661,176.507,15.244,151.955
C06828=1099.374,63.051,442.645,176.509,15.244,151.955
C06829=1099.380,63.300,442.629,176.512,15.245,151.954
C06830=1099.386,63.574,442.610,176.515,15.245,151.954
C06831=1099.393,63.847,442.592,176.518,15.246,151.953
C06832=1099.400,64.120,442.574,176.521,15.247,151.953
C06833=1099.405,64.394,442.556,176.523,15.247,151.952
C06834=1099.411,64.643,442.540,176.526,15.248,151.952
C06835=1099.417,64.892,442.522,176.528,15.248,151.952
C06836=1099.423,65.142,442.506,176.531,15.248,151.951
C06837=1099.429,65.391,442.490,176.534,15.249,151.951
C06838=1099.434,65.641,442.473,176.536,15.249,151.950
C06839=1099.440,65.890,442.457,176.539,15.250,151.950
C06840=1099.445,66.140,442.440,176.541,15.251,151.949
C06841=1099.451,66.388,442.423,176.543,15.250,151.949
C06842=1099.457,66.638,442.406,176.546,15.251,151.948
C06843=1099.462,66.887,442.390,176.549,15.252,151.948
C06844=1099.468,67.137,442.374,176.551,15.252,151.948
C06845=1099.474,67.386,442.357,176.554,15.253,151.947
C06846=1099.480,67.635,442.340,176.556,15.253,151.947
C06847=1099.485,67.885,442.323,176.559,15.254,151.946
C06848=1099.491,68.134,442.307,176.561,15.254,151.946
C06849=1099.496,68.384,442.290,176.564,15.255,151.945
C06850=1099.503,68.632,442.273,176.566,15.255,151.945
C06851=1099.508,68.882,442.256,176.569,15.255,151.944
C06852=1099.514,69.131,442.240,176.572,15.256,151.944
C06853=1099.519,69.381,442.223,176.574,15.256,151.943
C06854=1099.525,69.630,442.206,176.577,15.257,151.943
C06855=1099.530,69.879,442.189,176.579,15.257,151.943
C06856=1099.537,70.130,442.172,176.581,15.257,151.942
C06857=1099.542,70.379,442.155,176.584,15.258,151.942
C06858=1099.548,70.628,442.138,176.587,15.258,151.941
C06859=1099.554,70.878,442.122,176.590,15.259,151.941
C06860=1099.559,71.127,442.104,176.592,15.259,151.940
C06861=1099.565,71.376,442.088,176.595,15.260,151.940
C06862=1099.570,71.626,442.071,176.597,15.261,151.939
C06863=1099.576,71.875,442.054,176.600,15.260,151.939
C06864=1099.582,72.124,442.037,176.603,15.261,151.938
C06865=1099.587,72.373,442.020,176.605,15.262,151.938
C06866=1099.593,72.622,442.003,176.608,15.263,151.938
C06867=1099.598,72.872,441.987,176.610,15.262,151.937
C06868=1099.605,73.122,441.969,176.613,15.263,151.937
C06869=1099.611,73.371,441.952,176.615,15.264,151.936
C06870=1099.616,73.620,441.935,176.618,15.264,151.936
C06871=1099.621,73.870,441.918,176.621,15.264,151.935
C06872=1099.627,74.119,441.901,176.623,15.265,151.935
C06873=1099.633,74.368,441.884,176.626,15.265,151.934
C06874=1099.638,74.617,441.867,176.629,15.265,151.934
C06875=1099.644,74.867,441.850,176.631,15.266,151.933
C06876=1099.650,75.116,441.832,176.634,15.267,151.933
C06877=1099.656,75.366,441.816,176.636,15.266,151.932
C06878=1099.662,75.615,441.799,176.639,15.267,151.932
C06879=1099.667,75.864,441.782,176.641,15.268,151.931
C06880=1099.672,76.113,441.764,176.645,15.268,151.931
C06881=1099.678,76.363,441.748,176.647,15.268,151.930
C06882=1099.684,76.612,441.730,176.649,15.269,151.930
C06883=1099.690,76.862,441.713,176.652,15.269,151.929
C06884=1099.696,77.111,441.696,176.654,15.269,151.929
C06885=1099.701,77.361,441.679,176.658,15.270,151.928
C06886=1099.707,77.610,441.662,176.660,15.270,151.928
C06887=1099.712,77.859,441.644,176.662,15.270,151.928
C06888=1099.719,78.109,441.628,176.665,15.271,151.927
C06889=1099.724,78.358,441.610,176.668,15.271,151.927
C06890=1099.730,78.607,441.593,176.671,15.272,151.926
C06891=1099.735,78.856,441.576,176.673,15.272,151.926
C06892=1099.741,79.105,441.558,176.676,15.272,151.925
C06893=1099.747,79.356,441.541,176.679,15.273,151.925
C06894=1099.753,79.629,441.522,176.682,15.273,151.924
C06895=1099.759,79.902,441.503,176.684,15.273,151.924
C06896=1099.765,80.175,441.484,176.687,15.274,151.923
C06897=1099.771,80.448,441.465,176.691,15.274,151.922
C06898=1099.777,80.697,441.448,176.693,15.275,151.922
C06899=1099.783,80.947,441.430,176.696,15.275,151.922
C06900=1099.788,81.197,441.413,176.698,15.275,151.921
C06901=1099.794,81.446,441.396,176.701,15.276,151.921
C06902=1099.799,81.695,441.378,176.704,15.276,151.920
C06903=1099.806,81.944,441.360,176.706,15.276,151.920
C06904=1099.811,82.194,441.343,176.709,15.277,151.919
C06905=1099.816,82.443,441.326,176.711,15.277,151.919
C06906=1099.822,82.692,441.308,176.715,15.278,151.918
C06907=1099.827,82.941,441.291,176.717,15.278,151.918
C06908=1099.833,83.192,441.274,176.720,15.278,151.917
C06909=1099.839,83.441,441.256,176.722,15.279,151.917
C06910=1099.845,83.689,441.239,176.725,15.279,151.916
C06911=1099.851,83.939,441.221,176.728,15.279,151.916
C06912=1099.856,84.188,441.204,176.730,15.279,151.915
C06913=1099.862,84.437,441.186,176.733,15.280,151.915
C06914=1099.867,84.687,441.169,176.736,15.280,151.914
C06915=1099.873,84.937,441.151,176.739,15.280,151.913
C06916=1099.879,85.186,441.134,176.741,15.281,151.913
C06917=1099.884,85.435,441.116,176.744,15.281,151.912
C06918=1099.891,85.684,441.098,176.747,15.281,151.912
C06919=1099.896,85.933,441.081,176.750,15.282,151.911
C06920=1099.902,86.182,441.063,176.752,15.282,151.911
C06921=1099.907,86.431,441.045,176.755,15.283,151.910
C06922=1099.913,86.682,441.028,176.758,15.283,151.910
C06923=1099.918,86.931,441.011,176.760,15.283,151.909
C06924=1099.924,87.180,440.993,176.763,15.283,151.909
C06925=1099.930,87.430,440.975,176.766,15.283,151.908
C06926=1099.936,87.679,440.958,176.769,15.284,151.908
C06927=1099.941,87.928,440.940,176.771,15.284,151.907
C06928=1099.947,88.178,440.922,176.774,15.284,151.907
C06929=1099.953,88.427,440.904,176.777,15.284,151.906
C06930=1099.959,88.676,440.887,176.780,15.285,151.906
C06931=1099.964,88.925,440.869,176.782,15.285,151.905
C06932=1099.970,89.174,440.851,176.786,15.285,151.904
C06933=1099.976,89.424,440.833,176.788,15.286,151.904
C06934=1099.982,89.673,440.816,176.790,15.286,151.903
C06935=1099.987,89.922,440.798,176.794,15.286,151.903
C06936=1099.993,90.172,440.780,176.796,15.286,151.902
C06937=1099.998,90.421,440.762,176.799,15.287,151.902
C06938=1100.004,90.670,440.744,176.802,15.287,151.901
C06939=1100.010,90.919,440.726,176.805,15.287,151.901
C06940=1100.015,91.168,440.708,176.807,15.287,151.900
C06941=1100.022,91.418,440.691,176.810,15.288,151.900
C06942=1100.027,91.667,440.673,176.813,15.288,151.899
C06943=1100.033,91.917,440.655,176.816,15.288,151.899
C06944=1100.038,92.166,440.637,176.819,15.288,151.898
C06945=1100.043,92.415,440.619,176.822,15.289,151.898
C06946=1100.050,92.665,440.601,176.824,15.289,151.897
C06947=1100.055,92.914,440.584,176.826,15.289,151.896
C06948=1100.060,93.163,440.565,176.830,15.289,151.896
C06949=1100.066,93.413,440.547,176.832,15.289,151.895
C06950=1100.072,93.662,440.529,176.835,15.290,151.895
C06951=1100.078,93.911,440.511,176.838,15.290,151.894
C06952=1100.083,94.161,440.493,176.841,15.290,151.894
C06953=1100.089,94.409,440.475,176.843,15.290,151.893
C06954=1100.095,94.659,440.457,176.846,15.291,151.893
C06955=1100.100,94.908,440.440,176.849,15.291,151.892
C06956=1100.106,95.158,440.421,176.852,15.291,151.891
C06957=1100.111,95.407,440.403,176.855,15.291,151.891
C06958=1100.118,95.680,440.383,176.858,15.292,151.890
C06959=1100.124,95.953,440.363,176.861,15.292,151.890
C06960=1100.130,96.227,440.344,176.864,15.292,151.889
C06961=1100.136,96.500,440.324,176.867,15.292,151.889
C06962=1100.142,96.750,440.306,176.870,15.293,151.888
C06963=1100.147,96.999,440.288,176.873,15.293,151.887
C06964=1100.153,97.248,440.269,176.875,15.293,151.887
C06965=1100.159,97.497,440.251,176.879,15.293,151.886
C06966=1100.165,97.747,440.233,176.881,15.293,151.886
C06967=1100.170,97.996,440.215,176.884,15.293,151.885
C06968=1100.176,98.245,440.197,176.887,15.293,151.884
C06969=1100.182,98.494,440.179,176.890,15.294,151.884
C06970=1100.187,98.744,440.160,176.893,15.293,151.883
C06971=1100.193,98.993,440.142,176.896,15.294,151.883
C06972=1100.199,99.242,440.124,176.898,15.294,151.882
C06973=1100.204,99.491,440.105,176.902,15.294,151.882
C06974=1100.210,99.741,440.088,176.904,15.294,151.881
C06975=1100.216,99.989,440.069,176.907,15.295,151.880
C06976=1100.221,100.240,440.051,176.910,15.294,151.880
C06977=1100.228,100.489,440.032,176.913,15.295,151.879
C06978=1100.233,100.738,440.014,176.916,15.295,151.879
C06979=1100.239,100.987,439.995,176.919,15.295,151.878
C06980=1100.245,101.236,439.978,176.921,15.295,151.877
C06981=1100.250,101.486,439.958,176.925,15.296,151.877
C06982=1100.256,101.735,439.941,176.927,15.295,151.876
C06983=1100.262,101.984,439.922,176.930,15.296,151.876
C06984=1100.267,102.233,439.904,176.933,15.296,151.875
C06985=1100.273,102.483,439.885,176.936,15.296,151.875
C06986=1100.278,102.732,439.867,176.939,15.296,151.874
C06987=1100.284,102.981,439.848,176.942,15.297,151.873
C06988=1100.289,103.230,439.830,176.944,15.296,151.873
C06989=1100.295,103.480,439.811,176.948,15.297,151.872
C06990=1100.301,103.729,439.793,176.950,15.297,151.872
C06991=1100.306,103.978,439.774,176.953,15.297,151.871
C06992=1100.312,104.228,439.756,176.956,15.297,151.871
C06993=1100.318,104.476,439.738,176.960,15.297,151.870
C06994=1100.323,104.726,439.718,176.962,15.297,151.869
C06995=1100.329,104.975,439.701,176.965,15.297,151.869
C06996=1100.334,105.224,439.682,176.968,15.297,151.868
C06997=1100.341,105.474,439.664,176.971,15.298,151.867
C06998=1100.346,105.723,439.645,176.974,15.298,151.867
C06999=1100.351,105.972,439.626,176.977,15.298,151.866
C07000=1100.357,106.221,439.608,176.979,15.298,151.866
C07001=1100.363,106.471,439.589,176.983,15.298,151.865
C07002=1100.369,106.720,439.570,176.985,15.298,151.864
C07003=1100.374,106.969,439.552,176.989,15.298,151.864
C07004=1100.379,107.219,439.533,176.991,15.298,151.863
C07005=1100.386,107.468,439.514,176.994,15.299,151.863
C07006=1100.391,107.716,439.495,176.997,15.298,151.862
C07007=1100.397,107.966,439.477,177.001,15.299,151.861
C07008=1100.402,108.215,439.458,177.003,15.298,151.861
C07009=1100.408,108.464,439.439,177.006,15.299,151.860
C07010=1100.414,108.714,439.421,177.009,15.299,151.860
C07011=1100.419,108.963,439.402,177.012,15.299,151.859
C07012=1100.425,109.212,439.384,177.015,15.299,151.858
C07013=1100.431,109.461,439.364,177.018,15.299,151.858
C07014=1100.437,109.711,439.345,177.021,15.298,151.857
C07015=1100.442,109.960,439.328,177.024,15.299,151.856
C07016=1100.448,110.209,439.308,177.027,15.299,151.856
C07017=1100.454,110.459,439.289,177.030,15.299,151.855
C07018=1100.460,110.707,439.271,177.033,15.299,151.854
C07019=1100.465,110.957,439.252,177.036,15.299,151.854
C07020=1100.471,111.206,439.232,177.039,15.299,151.853
C07021=1100.476,111.455,439.215,177.042,15.299,151.853
C07022=1100.483,111.728,439.193,177.045,15.299,151.852
C07023=1100.489,112.002,439.172,177.048,15.299,151.851
C07024=1100.495,112.275,439.152,177.052,15.299,151.850
C07025=1100.501,112.549,439.131,177.055,15.299,151.850
C07026=1100.507,112.798,439.112,177.058,15.299,151.849
C07027=1100.513,113.048,439.093,177.061,15.299,151.849
C07028=1100.518,113.296,439.074,177.064,15.299,151.848
C07029=1100.524,113.546,439.055,177.067,15.299,151.847
C07030=1100.530,113.795,439.036,177.070,15.299,151.847
C07031=1100.535,114.044,439.018,177.073,15.299,151.846
C07032=1100.541,114.293,438.998,177.076,15.299,151.845
C07033=1100.547,114.542,438.979,177.079,15.300,151.845
C07034=1100.553,114.792,438.960,177.082,15.299,151.844
C07035=1100.558,115.041,438.941,177.085,15.299,151.843
C07036=1100.563,115.290,438.922,177.088,15.299,151.843
C07037=1100.569,115.539,438.902,177.091,15.299,151.842
C07038=1100.575,115.789,438.883,177.094,15.299,151.842
C07039=1100.580,116.038,438.864,177.097,15.299,151.841
C07040=1100.585,116.287,438.845,177.100,15.299,151.840
C07041=1100.591,116.537,438.826,177.103,15.300,151.840
C07042=1100.596,116.785,438.807,177.106,15.299,151.839
C07043=1100.602,117.035,438.788,177.109,15.299,151.838
C07044=1100.608,117.284,438.768,177.113,15.300,151.838
C07045=1100.613,117.534,438.749,177.115,15.299,151.837
C07046=1100.618,117.782,438.730,177.118,15.300,151.836
C07047=1100.624,118.032,438.711,177.121,15.299,151.836
C07048=1100.630,118.281,438.691,177.124,15.300,151.835
C07049=1100.636,118.530,438.672,177.127,15.299,151.834
C07050=1100.641,118.779,438.653,177.131,15.300,151.834
C07051=1100.647,119.028,438.634,177.133,15.299,151.833
C07052=1100.652,119.278,438.615,177.137,15.300,151.832
C07053=1100.658,119.527,438.595,177.139,15.299,151.832
C07054=1100.664,119.776,438.575,177.143,15.300,151.831
C07055=1100.670,120.025,438.556,177.145,15.299,151.830
C07056=1100.675,120.274,438.537,177.149,15.299,151.830
C07057=1100.680,120.523,438.518,177.152,15.299,151.829
C07058=1100.686,120.773,438.499,177.155,15.299,151.828
C07059=1100.692,121.022,438.479,177.158,15.299,151.828
C07060=1100.698,121.271,438.460,177.161,15.299,151.827
C07061=1100.703,121.521,438.440,177.164,15.299,151.826
C07062=1100.708,121.769,438.421,177.167,15.299,151.826
C07063=1100.714,122.018,438.401,177.171,15.299,151.825
C07064=1100.720,122.267,438.382,177.173,15.299,151.824
C07065=1100.726,122.517,438.363,177.177,15.299,151.824
C07066=1100.732,122.766,438.343,177.179,15.299,151.823
C07067=1100.738,123.015,438.324,177.183,15.299,151.822
C07068=1100.743,123.265,438.305,177.186,15.298,151.822
C07069=1100.748,123.513,438.284,177.189,15.298,151.821
C07070=1100.754,123.762,438.265,177.192,15.298,151.820
C07071=1100.759,124.012,438.246,177.195,15.298,151.820
C07072=1100.765,124.261,438.226,177.198,15.298,151.819
C07073=1100.771,124.510,438.207,177.202,15.298,151.818
C07074=1100.777,124.760,438.187,177.205,15.298,151.817
C07075=1100.783,125.008,438.167,177.208,15.298,151.817
C07076=1100.788,125.258,438.148,177.211,15.298,151.816
C07077=1100.794,125.507,438.128,177.214,15.297,151.815
C07078=1100.799,125.756,438.108,177.218,15.297,151.815
C07079=1100.805,126.006,438.089,177.220,15.297,151.814
C07080=1100.811,126.255,438.069,177.224,15.297,151.813
C07081=1100.817,126.504,438.050,177.226,15.297,151.813
C07082=1100.823,126.753,438.030,177.230,15.297,151.812
C07083=1100.828,127.002,438.011,177.233,15.296,151.811
C07084=1100.834,127.250,437.991,177.236,15.297,151.811
C07085=1100.839,127.500,437.971,177.239,15.296,151.810
C07086=1100.846,127.774,437.950,177.242,15.296,151.809
C07087=1100.852,128.047,437.928,177.246,15.296,151.808
C07088=1100.858,128.320,437.906,177.250,15.296,151.807
C07089=1100.864,128.593,437.885,177.253,15.296,151.807
C07090=1100.870,128.843,437.865,177.256,15.295,151.806
C07091=1100.876,129.091,437.845,177.260,15.295,151.805
C07092=1100.882,129.340,437.825,177.263,15.295,151.805
C07093=1100.887,129.590,437.806,177.266,15.295,151.804
C07094=1100.893,129.840,437.785,177.269,15.295,151.803
C07095=1100.899,130.089,437.766,177.272,15.295,151.802
C07096=1100.905,130.338,437.746,177.275,15.294,151.802
C07097=1100.910,130.587,437.725,177.279,15.294,151.801
C07098=1100.916,130.836,437.706,177.282,15.294,151.800
C07099=1100.922,131.085,437.686,177.285,15.294,151.799
C07100=1100.928,131.334,437.666,177.289,15.294,151.799
C07101=1100.934,131.583,437.647,177.291,15.293,151.798
C07102=1100.939,131.833,437.627,177.295,15.293,151.797
C07103=1100.945,132.081,437.607,177.298,15.293,151.797
C07104=1100.950,132.331,437.587,177.301,15.293,151.796
C07105=1100.956,132.580,437.567,177.304,15.292,151.795
C07106=1100.962,132.829,437.547,177.308,15.292,151.794
C07107=1100.967,133.078,437.526,177.311,15.292,151.794
C07108=1100.973,133.327,437.507,177.314,15.292,151.793
C07109=1100.979,133.576,437.487,177.317,15.291,151.792
C07110=1100.984,133.825,437.466,177.321,15.291,151.791
C07111=1100.990,134.074,437.447,177.324,15.291,151.791
C07112=1100.995,134.324,437.427,177.327,15.291,151.790
C07113=1101.001,134.573,437.407,177.331,15.291,151.789
C07114=1101.007,134.822,437.386,177.333,15.290,151.788
C07115=1101.013,135.071,437.366,177.337,15.290,151.788
C07116=1101.019,135.320,437.346,177.340,15.290,151.787
C07117=1101.024,135.570,437.326,177.343,15.290,151.786
C07118=1101.030,135.819,437.306,177.346,15.289,151.785
C07119=1101.035,136.068,437.286,177.350,15.289,151.785
C07120=1101.041,136.316,437.266,177.353,15.289,151.784
C07121=1101.046,136.566,437.245,177.356,15.289,151.783
C07122=1101.052,136.814,437.225,177.360,15.289,151.783
C07123=1101.057,137.064,437.205,177.362,15.288,151.782
C07124=1101.064,137.314,437.185,177.366,15.288,151.781
C07125=1101.069,137.563,437.164,177.369,15.288,151.780
C07126=1101.075,137.812,437.144,177.372,15.288,151.780
C07127=1101.080,138.061,437.124,177.376,15.288,151.779
C07128=1101.086,138.310,437.104,177.379,15.287,151.778
C07129=1101.091,138.559,437.083,177.383,15.287,151.777
C07130=1101.097,138.807,437.063,177.385,15.286,151.776
C07131=1101.103,139.057,437.042,177.389,15.286,151.776
C07132=1101.109,139.306,437.022,177.392,15.286,151.775
C07133=1101.115,139.555,437.002,177.395,15.286,151.774
C07134=1101.120,139.804,436.981,177.398,15.285,151.774
C07135=1101.126,140.053,436.961,177.402,15.286,151.773
C07136=1101.131,140.302,436.941,177.406,15.285,151.772
C07137=1101.138,140.552,436.921,177.408,15.285,151.771
C07138=1101.143,140.801,436.900,177.412,15.285,151.770
C07139=1101.148,141.050,436.879,177.415,15.284,151.770
C07140=1101.154,141.299,436.859,177.418,15.284,151.769
C07141=1101.159,141.548,436.839,177.421,15.284,151.768
C07142=1101.165,141.797,436.818,177.425,15.283,151.767
C07143=1101.171,142.047,436.798,177.429,15.283,151.767
C07144=1101.177,142.295,436.777,177.431,15.283,151.766
C07145=1101.182,142.544,436.756,177.435,15.283,151.765
C07146=1101.188,142.793,436.736,177.438,15.282,151.764
C07147=1101.193,143.042,436.716,177.442,15.282,151.763
C07148=1101.199,143.291,436.695,177.445,15.281,151.763
C07149=1101.204,143.541,436.674,177.448,15.281,151.762
C07150=1101.211,143.814,436.652,177.452,15.281,151.761
C07151=1101.217,144.088,436.629,177.456,15.281,151.760
C07152=1101.223,144.360,436.607,177.459,15.281,151.759
C07153=1101.230,144.634,436.584,177.463,15.280,151.759
C07154=1101.235,144.883,436.563,177.466,15.280,151.758
C07155=1101.240,145.132,436.543,177.470,15.279,151.757
C07156=1101.246,145.381,436.523,177.473,15.279,151.756
C07157=1101.252,145.630,436.501,177.476,15.279,151.755
C07158=1101.258,145.879,436.480,177.480,15.278,151.755
C07159=1101.263,146.128,436.460,177.483,15.278,151.754
C07160=1101.269,146.376,436.439,177.486,15.278,151.753
C07161=1101.275,146.626,436.418,177.490,15.277,151.752
C07162=1101.280,146.875,436.398,177.493,15.277,151.751
C07163=1101.286,147.124,436.377,177.496,15.276,151.751
C07164=1101.292,147.374,436.356,177.500,15.276,151.750
C07165=1101.298,147.623,436.336,177.503,15.276,151.749
C07166=1101.303,147.872,436.315,177.507,15.275,151.748
C07167=1101.309,148.121,436.293,177.510,15.275,151.747
C07168=1101.314,148.370,436.273,177.513,15.275,151.747
C07169=1101.320,148.619,436.252,177.517,15.275,151.746
C07170=1101.325,148.868,436.231,177.520,15.274,151.745
C07171=1101.332,149.117,436.211,177.524,15.274,151.744
C07172=1101.337,149.366,436.189,177.527,15.273,151.743
C07173=1101.343,149.615,436.169,177.530,15.273,151.743
C07174=1101.349,149.865,436.148,177.534,15.273,151.742
C07175=1101.354,150.113,436.127,177.537,15.272,151.741
C07176=1101.359,150.362,436.106,177.541,15.272,151.740
C07177=1101.366,150.611,436.085,177.544,15.271,151.739
C07178=1101.371,150.861,436.064,177.547,15.271,151.739
C07179=1101.376,151.109,436.043,177.550,15.271,151.738
C07180=1101.382,151.359,436.022,177.554,15.270,151.737
C07181=1101.388,151.607,436.001,177.558,15.270,151.736
C07182=1101.393,151.856,435.980,177.561,15.269,151.735
C07183=1101.399,152.106,435.958,177.564,15.269,151.735
C07184=1101.404,152.355,435.938,177.567,15.268,151.734
C07185=1101.410,152.603,435.917,177.571,15.269,151.733
C07186=1101.416,152.853,435.896,177.575,15.268,151.732
C07187=1101.421,153.102,435.874,177.578,15.267,151.731
C07188=1101.427,153.351,435.853,177.582,15.267,151.730
C07189=1101.433,153.600,435.832,177.585,15.266,151.729
C07190=1101.438,153.848,435.811,177.588,15.266,151.729
C07191=1101.444,154.098,435.790,177.592,15.266,151.728
C07192=1101.450,154.347,435.769,177.595,15.265,151.727
C07193=1101.456,154.596,435.747,177.599,15.265,151.726
C07194=1101.461,154.845,435.727,177.602,15.264,151.725
C07195=1101.467,155.094,435.705,177.605,15.264,151.725
C07196=1101.473,155.343,435.684,177.609,15.264,151.724
C07197=1101.478,155.592,435.663,177.612,15.263,151.723
C07198=1101.484,155.841,435.641,177.616,15.263,151.722
C07199=1101.490,156.090,435.621,177.619,15.262,151.721
C07200=1101.496,156.339,435.599,177.623,15.262,151.720
C07201=1101.501,156.588,435.577,177.627,15.262,151.719
C07202=1101.506,156.837,435.556,177.630,15.261,151.719
C07203=1101.512,157.087,435.535,177.633,15.261,151.718
C07204=1101.518,157.335,435.514,177.636,15.260,151.717
C07205=1101.524,157.584,435.492,177.640,15.260,151.716
C07206=1101.529,157.833,435.471,177.644,15.260,151.715
C07207=1101.535,158.083,435.450,177.647,15.259,151.714
C07208=1101.540,158.331,435.428,177.651,15.258,151.714
C07209=1101.546,158.581,435.407,177.654,15.258,151.713
C07210=1101.552,158.829,435.385,177.658,15.258,151.712
C07211=1101.558,159.078,435.364,177.661,15.257,151.711
C07212=1101.563,159.328,435.343,177.665,15.256,151.710
C07213=1101.569,159.577,435.321,177.668,15.256,151.709
C07214=1101.575,159.849,435.298,177.672,15.256,151.708
C07215=1101.581,160.123,435.274,177.675,15.255,151.707
C07216=1101.587,160.395,435.251,177.679,15.254,151.707
C07217=1101.593,160.668,435.227,177.683,15.254,151.706
C07218=1101.600,160.918,435.205,177.687,15.254,151.705
C07219=1101.605,161.166,435.184,177.690,15.253,151.704
C07220=1101.611,161.416,435.162,177.694,15.252,151.703
C07221=1101.616,161.664,435.141,177.698,15.252,151.702
C07222=1101.622,161.913,435.119,177.701,15.251,151.701
C07223=1101.627,162.162,435.097,177.705,15.251,151.700
C07224=1101.633,162.411,435.076,177.708,15.250,151.700
C07225=1101.639,162.660,435.054,177.711,15.250,151.699
C07226=1101.644,162.909,435.032,177.715,15.250,151.698
C07227=1101.650,163.158,435.011,177.718,15.249,151.697
C07228=1101.655,163.407,434.989,177.722,15.249,151.696
C07229=1101.661,163.656,434.967,177.726,15.249,151.695
C07230=1101.666,163.905,434.945,177.729,15.248,151.694
C07231=1101.672,164.154,434.924,177.733,15.247,151.694
C07232=1101.677,164.403,434.902,177.736,15.246,151.693
C07233=1101.683,164.652,434.880,177.740,15.247,151.692
C07234=1101.688,164.901,434.858,177.743,15.246,151.691
C07235=1101.694,165.150,434.837,177.747,15.245,151.690
C07236=1101.699,165.399,434.815,177.750,15.245,151.689
C07237=1101.705,165.648,434.793,177.754,15.245,151.688
C07238=1101.710,165.897,434.771,177.757,15.244,151.687
C07239=1101.716,166.146,434.750,177.761,15.244,151.687
C07240=1101.721,166.395,434.728,177.764,15.243,151.686
C07241=1101.727,166.644,434.706,177.768,15.242,151.685
C07242=1101.732,166.893,434.683,177.772,15.242,151.684
C07243=1101.739,167.142,434.662,177.775,15.241,151.683
C07244=1101.743,167.391,434.640,177.779,15.241,151.682
C07245=1101.750,167.640,434.618,177.783,15.241,151.681
C07246=1101.754,167.889,434.596,177.786,15.240,151.680
C07247=1101.761,168.138,434.575,177.790,15.239,151.680
C07248=1101.766,168.387,434.552,177.793,15.238,151.679
C07249=1101.772,168.635,434.530,177.796,15.238,151.678
C07250=1101.777,168.885,434.508,177.800,15.238,151.677
C07251=1101.783,169.134,434.487,177.803,15.237,151.676
C07252=1101.789,169.382,434.464,177.807,15.237,151.675
C07253=1101.794,169.632,434.442,177.811,15.237,151.674
C07254=1101.800,169.880,434.421,177.814,15.236,151.674
C07255=1101.805,170.130,434.398,177.818,15.235,151.673
C07256=1101.812,170.379,434.376,177.821,15.234,151.672
C07257=1101.816,170.627,434.354,177.825,15.234,151.671
C07258=1101.822,170.877,434.332,177.829,15.234,151.670
C07259=1101.828,171.125,434.310,177.832,15.233,151.669
C07260=1101.833,171.374,434.288,177.836,15.232,151.668
C07261=1101.839,171.623,434.266,177.840,15.232,151.667
C07262=1101.845,171.872,434.243,177.843,15.231,151.666
C07263=1101.850,172.121,434.221,177.847,15.230,151.665
C07264=1101.856,172.370,434.199,177.851,15.230,151.664
C07265=1101.862,172.619,434.177,177.854,15.229,151.664
C07266=1101.867,172.869,434.154,177.858,15.229,151.663
C07267=1101.873,173.117,434.132,177.861,15.228,151.662
C07268=1101.878,173.366,434.110,177.865,15.228,151.661
